		//Check for error after read request
		IF NOT fbADSREADWRITE_ReadAds.BUSY AND NOT fbADSREADWRITE_ReadAds.ERR AND byCounterWaitInStep_ReadAds >= byStaticValueWaitInStep THEN 
			IF udiNumberSizeValues_ReadAds >= 1 AND udiNumberSizeValues_ReadAds <= 4000 THEN
				FOR udiLPCheckErrorAfterReadReq_ReadAds := 1 TO (udiNumberSizeValues_ReadAds * 4) BY 1 DO
					IF arrValueRead_ReadAds[udiLPCheckErrorAfterReadReq_ReadAds] <> 0 THEN iState_ReadAds := 200; EXIT; END_IF
				END_FOR
			END_IF
		END_IF 	
	
		IF NOT fbADSREADWRITE_ReadAds.BUSY AND NOT fbADSREADWRITE_ReadAds.ERR AND byCounterWaitInStep_ReadAds >= byStaticValueWaitInStep AND iState_ReadAds = -5 THEN 
			byCounterWaitInStep_ReadAds := 0;	
				fbADSREADWRITE_ReadAds.WRTRD := FALSE;
				 iState_ReadAds := -4;
				 	udiStartValueReadOutReqBuffer_AdsRead := (udiNumberSizeValues_ReadAds * 4) + 1;	
						udiNumberInProgress_ReadAds := 1;
		 END_IF 
		
			IF FPErrorReadWrite_ReadAds.Q OR timTimout_ReadAds.Q THEN iState_ReadAds := 200; END_IF 	
			
	-4://Copy Value in buffer after read request and clear data
		uiNumberValueSymbolSize_ReadAds := 0; byNumberOfValues_ReadAds_ReadAds := 0; byLenghSymbolName_ReadAds := 0; byValueInTurn_ReadAds := 0; byCounterValue_ReadAds	:= 0;
			uiValueForLoopStart_ReadAds := 0; uiValueForLoopStop_ReadAds := 0; byCounterValueReadOut_ReadAds := 0;
				fbADSREADWRITE_ReadAds.WRTRD := FALSE;	
		arrCounterWriteValueInArray_ReadAds[1] := 0; arrCounterWriteValueInArray_ReadAds[2] := 0; arrCounterWriteValueInArray_ReadAds[3] := 0; arrCounterWriteValueInArray_ReadAds[4] := 0; arrCounterWriteValueInArray_ReadAds[5] := 0;
			arrCounterWriteValueInArray_ReadAds[6] := 0; arrCounterWriteValueInArray_ReadAds[7] := 0; arrCounterWriteValueInArray_ReadAds[8] := 0;
									
		uiCounterArrayOfString_ReadAds := 0;
	
		sStringFloat_ReadAds := ''; iFindPointFloat_ReadAds := 0; iPrecision_ReadAds := 0;
		
		//Copy first 800 default bytes to save resources on small plc's
		MEMCPY(ADR(arrValueAfterRead_ReadAds),ADR(arrValueAfterReadDefault_ReadAds),SIZEOF(arrValueAfterRead_ReadAds));
		
		//Clear lengh from each value
		arrLenghEachValue_ReadAds := arrLenghEachValueDefault_ReadAds;
			
		//Clear array with symbol name and array with the value names
		arrSymbolName_ReadAds := arrSymbolNameDefault_ReadAds;
			arrValueName_ReadAds := arrValueNameDefault_ReadAds; 
	
		//Copy the values
		udiNumberInProgress_ReadAds := LIMIT(1,udiNumberInProgress_ReadAds,10);
			udiStopValueReadOutReqBuffer_AdsRead := (udiStartValueReadOutReqBuffer_AdsRead - 1) + arrInfoValue_Read_Ads[udiNumberInProgress_ReadAds].udiLength;

		IF udiStartValueReadOutReqBuffer_AdsRead >= 1 AND udiStartValueReadOutReqBuffer_AdsRead <= 1600 AND udiStopValueReadOutReqBuffer_AdsRead >= 1 AND udiStopValueReadOutReqBuffer_AdsRead <= 1600 THEN  
			FOR udiLPCopyValueFromReqBuffer_ReadAds := udiStartValueReadOutReqBuffer_AdsRead TO udiStopValueReadOutReqBuffer_AdsRead BY 1 DO
				uiCounterCopyValueFromReqBuffer_ReadAds := LIMIT(1,uiCounterCopyValueFromReqBuffer_ReadAds,1600);	
					arrValueAfterRead_ReadAds[uiCounterCopyValueFromReqBuffer_ReadAds] := arrValueRead_ReadAds[udiLPCopyValueFromReqBuffer_ReadAds]; 
						uiCounterCopyValueFromReqBuffer_ReadAds := uiCounterCopyValueFromReqBuffer_ReadAds + 1;
			END_FOR 
		END_IF		
			
		uiCounterCopyValueFromReqBuffer_ReadAds := 0;
			udiActiveNumberOfSymbol_ReadAds := udiActiveNumberOfSymbol_ReadAds + 1;
				udiActiveNumberOfSymbol_ReadAds := LIMIT(1,udiActiveNumberOfSymbol_ReadAds,Lynus_Standards.Constants_Communicator.udiArraySizeMarkedSymobls);
					udiStartValueReadOutReqBuffer_AdsRead := udiStopValueReadOutReqBuffer_AdsRead + 1;
						iState_ReadAds := -3;
						
	-3://Check whether the write application does not have the same value as when reading
		IF (Lynus_Standards.GVL_Communicator.arrInterfaceInfoAlVariables[byReadWriteArrayNumber,udiActiveNumberOfSymbol_ReadAds].sFullSymbolName <> Lynus_Standards.GVL_Communicator.arrInterfaceInfoValueWriteTo[byReadWriteArrayNumber].sFullSymbolName) 
			// AND m_EnableChange_upload) // Stefan added AND 
			// OR m_TriggerIntervalSend=TRUE THEN 	// STEFAN
			THEN
			iState_ReadAds := 5;
		ELSE
			IF udiActiveNumberOfSymbol_ReadAds < Lynus_Standards.GVL_Communicator.arrCounterVariableInArray[byReadWriteArrayNumber] AND udiNumberInProgress_ReadAds < udiNumberSizeValues_ReadAds THEN iState_ReadAds := -4; udiNumberInProgress_ReadAds := udiNumberInProgress_ReadAds + 1; END_IF
			IF (udiNumberInProgress_ReadAds >= udiNumberSizeValues_ReadAds AND iState_ReadAds = -3) THEN iState_ReadAds := -8; udiNumberInProgress_ReadAds := 0; END_IF
			IF udiActiveNumberOfSymbol_ReadAds >= Lynus_Standards.GVL_Communicator.arrCounterVariableInArray[byReadWriteArrayNumber] THEN iState_ReadAds := -8; udiActiveNumberOfSymbol_ReadAds := 0; udiNumberInProgress_ReadAds := 0; udiRestValueSymbolRead_ReadAds := 0; END_IF 
		END_IF  
	
		//Timeout
		IF timTimout_ReadAds.Q THEN iState_ReadAds := 200; END_IF
		
	5://Write value and symbol name in read array
	
		IF (Lynus_Standards.GVL_Communicator.arrInterfaceInfoAlVariables[byReadWriteArrayNumber,udiActiveNumberOfSymbol_ReadAds].sFullSymbolName <> Lynus_Standards.GVL_Communicator.arrInterfaceInfoValueWriteTo[byReadWriteArrayNumber].sFullSymbolName)
			// AND m_EnableChange_upload) // Stefan added AND 
			// OR m_TriggerIntervalSend=TRUE THEN 	// STEFAN
			THEN
			//Type BOOL
			IF Lynus_Standards.GVL_Communicator.arrInterfaceInfoAlVariables[byReadWriteArrayNumber,udiActiveNumberOfSymbol_ReadAds].sSymbolType = 'BOOL' THEN 
				stADSRead_ReadAds[udiActiveNumberOfSymbol_ReadAds].arrValue := arrValueDefault_ReadAds;
					stADSRead_ReadAds[udiActiveNumberOfSymbol_ReadAds].sFullSymbolName := Lynus_Standards.GVL_Communicator.arrInterfaceInfoAlVariables[byReadWriteArrayNumber,udiActiveNumberOfSymbol_ReadAds].sFullSymbolName; 
						stADSRead_ReadAds[udiActiveNumberOfSymbol_ReadAds].arrValue[1] := BYTE_TO_STRING(arrValueAfterRead_ReadAds[1]); 
			END_IF
				//Type BYTE
				IF Lynus_Standards.GVL_Communicator.arrInterfaceInfoAlVariables[byReadWriteArrayNumber,udiActiveNumberOfSymbol_ReadAds].sSymbolType = 'BYTE' THEN 
					stADSRead_ReadAds[udiActiveNumberOfSymbol_ReadAds].arrValue := arrValueDefault_ReadAds;
						stADSRead_ReadAds[udiActiveNumberOfSymbol_ReadAds].sFullSymbolName := Lynus_Standards.GVL_Communicator.arrInterfaceInfoAlVariables[byReadWriteArrayNumber,udiActiveNumberOfSymbol_ReadAds].sFullSymbolName; 
							stADSRead_ReadAds[udiActiveNumberOfSymbol_ReadAds].arrValue[1] := BYTE_TO_STRING(arrValueAfterRead_ReadAds[1]); 
				END_IF
			//Type WORD
			IF Lynus_Standards.GVL_Communicator.arrInterfaceInfoAlVariables[byReadWriteArrayNumber,udiActiveNumberOfSymbol_ReadAds].sSymbolType = 'WORD' THEN 
				stADSRead_ReadAds[udiActiveNumberOfSymbol_ReadAds].arrValue := arrValueDefault_ReadAds;
					stADSRead_ReadAds[udiActiveNumberOfSymbol_ReadAds].sFullSymbolName := Lynus_Standards.GVL_Communicator.arrInterfaceInfoAlVariables[byReadWriteArrayNumber,udiActiveNumberOfSymbol_ReadAds].sFullSymbolName; 
						stADSRead_ReadAds[udiActiveNumberOfSymbol_ReadAds].arrValue[1] := WORD_TO_STRING(SHL(BYTE_TO_WORD(arrValueAfterRead_ReadAds[2]),8) + BYTE_TO_WORD(arrValueAfterRead_ReadAds[1]));
			END_IF
				//Type DWORD
				IF Lynus_Standards.GVL_Communicator.arrInterfaceInfoAlVariables[byReadWriteArrayNumber,udiActiveNumberOfSymbol_ReadAds].sSymbolType = 'DWORD' THEN 
					stADSRead_ReadAds[udiActiveNumberOfSymbol_ReadAds].arrValue := arrValueDefault_ReadAds;
						stADSRead_ReadAds[udiActiveNumberOfSymbol_ReadAds].sFullSymbolName := Lynus_Standards.GVL_Communicator.arrInterfaceInfoAlVariables[byReadWriteArrayNumber,udiActiveNumberOfSymbol_ReadAds].sFullSymbolName; 
							stADSRead_ReadAds[udiActiveNumberOfSymbol_ReadAds].arrValue[1] := DWORD_TO_STRING(SHL(BYTE_TO_DWORD(arrValueAfterRead_ReadAds[4]),24) + SHL(BYTE_TO_DWORD(arrValueAfterRead_ReadAds[3]),16) + SHL(BYTE_TO_DWORD(arrValueAfterRead_ReadAds[2]),8) + BYTE_TO_DWORD(arrValueAfterRead_ReadAds[1]));
				END_IF
			//Type SINT
			IF Lynus_Standards.GVL_Communicator.arrInterfaceInfoAlVariables[byReadWriteArrayNumber,udiActiveNumberOfSymbol_ReadAds].sSymbolType = 'SINT' THEN 
				stADSRead_ReadAds[udiActiveNumberOfSymbol_ReadAds].arrValue := arrValueDefault_ReadAds;
					stADSRead_ReadAds[udiActiveNumberOfSymbol_ReadAds].sFullSymbolName := Lynus_Standards.GVL_Communicator.arrInterfaceInfoAlVariables[byReadWriteArrayNumber,udiActiveNumberOfSymbol_ReadAds].sFullSymbolName; 
						stADSRead_ReadAds[udiActiveNumberOfSymbol_ReadAds].arrValue[1] := SINT_TO_STRING(BYTE_TO_SINT(arrValueAfterRead_ReadAds[1]));
			END_IF
				//Type USINT
				IF Lynus_Standards.GVL_Communicator.arrInterfaceInfoAlVariables[byReadWriteArrayNumber,udiActiveNumberOfSymbol_ReadAds].sSymbolType = 'USINT' THEN 
					stADSRead_ReadAds[udiActiveNumberOfSymbol_ReadAds].arrValue := arrValueDefault_ReadAds;
						stADSRead_ReadAds[udiActiveNumberOfSymbol_ReadAds].sFullSymbolName := Lynus_Standards.GVL_Communicator.arrInterfaceInfoAlVariables[byReadWriteArrayNumber,udiActiveNumberOfSymbol_ReadAds].sFullSymbolName; 
							stADSRead_ReadAds[udiActiveNumberOfSymbol_ReadAds].arrValue[1] := USINT_TO_STRING(BYTE_TO_USINT(arrValueAfterRead_ReadAds[1]));
				END_IF
			//Type INT
			IF Lynus_Standards.GVL_Communicator.arrInterfaceInfoAlVariables[byReadWriteArrayNumber,udiActiveNumberOfSymbol_ReadAds].sSymbolType = 'INT' THEN 
				stADSRead_ReadAds[udiActiveNumberOfSymbol_ReadAds].arrValue := arrValueDefault_ReadAds;
					stADSRead_ReadAds[udiActiveNumberOfSymbol_ReadAds].sFullSymbolName := Lynus_Standards.GVL_Communicator.arrInterfaceInfoAlVariables[byReadWriteArrayNumber,udiActiveNumberOfSymbol_ReadAds].sFullSymbolName; 
						stADSRead_ReadAds[udiActiveNumberOfSymbol_ReadAds].arrValue[1] := INT_TO_STRING(SHL(BYTE_TO_INT(arrValueAfterRead_ReadAds[2]),8) + BYTE_TO_INT(arrValueAfterRead_ReadAds[1]));
			END_IF
				//Type UINT
				IF Lynus_Standards.GVL_Communicator.arrInterfaceInfoAlVariables[byReadWriteArrayNumber,udiActiveNumberOfSymbol_ReadAds].sSymbolType = 'UINT' THEN 
					stADSRead_ReadAds[udiActiveNumberOfSymbol_ReadAds].arrValue := arrValueDefault_ReadAds;
						stADSRead_ReadAds[udiActiveNumberOfSymbol_ReadAds].sFullSymbolName := Lynus_Standards.GVL_Communicator.arrInterfaceInfoAlVariables[byReadWriteArrayNumber,udiActiveNumberOfSymbol_ReadAds].sFullSymbolName; 
							stADSRead_ReadAds[udiActiveNumberOfSymbol_ReadAds].arrValue[1] := UINT_TO_STRING(SHL(BYTE_TO_UINT(arrValueAfterRead_ReadAds[2]),8) + BYTE_TO_UINT(arrValueAfterRead_ReadAds[1]));
				END_IF
			//Type DINT
			IF Lynus_Standards.GVL_Communicator.arrInterfaceInfoAlVariables[byReadWriteArrayNumber,udiActiveNumberOfSymbol_ReadAds].sSymbolType = 'DINT' THEN 
				stADSRead_ReadAds[udiActiveNumberOfSymbol_ReadAds].arrValue := arrValueDefault_ReadAds;
					stADSRead_ReadAds[udiActiveNumberOfSymbol_ReadAds].sFullSymbolName := Lynus_Standards.GVL_Communicator.arrInterfaceInfoAlVariables[byReadWriteArrayNumber,udiActiveNumberOfSymbol_ReadAds].sFullSymbolName; 
						stADSRead_ReadAds[udiActiveNumberOfSymbol_ReadAds].arrValue[1] := DINT_TO_STRING(SHL(BYTE_TO_DINT(arrValueAfterRead_ReadAds[4]),24) + SHL(BYTE_TO_DINT(arrValueAfterRead_ReadAds[3]),16) + SHL(BYTE_TO_DINT(arrValueAfterRead_ReadAds[2]),8) + BYTE_TO_DINT(arrValueAfterRead_ReadAds[1]));
			END_IF
				//Type UDINT
				IF Lynus_Standards.GVL_Communicator.arrInterfaceInfoAlVariables[byReadWriteArrayNumber,udiActiveNumberOfSymbol_ReadAds].sSymbolType = 'UDINT' THEN 
					stADSRead_ReadAds[udiActiveNumberOfSymbol_ReadAds].arrValue := arrValueDefault_ReadAds;
						stADSRead_ReadAds[udiActiveNumberOfSymbol_ReadAds].sFullSymbolName := Lynus_Standards.GVL_Communicator.arrInterfaceInfoAlVariables[byReadWriteArrayNumber,udiActiveNumberOfSymbol_ReadAds].sFullSymbolName; 
							stADSRead_ReadAds[udiActiveNumberOfSymbol_ReadAds].arrValue[1] := UDINT_TO_STRING(SHL(BYTE_TO_UDINT(arrValueAfterRead_ReadAds[4]),24) + SHL(BYTE_TO_UDINT(arrValueAfterRead_ReadAds[3]),16) + SHL(BYTE_TO_UDINT(arrValueAfterRead_ReadAds[2]),8) + BYTE_TO_UDINT(arrValueAfterRead_ReadAds[1]));
				END_IF
			//Type LINT
			IF Lynus_Standards.GVL_Communicator.arrInterfaceInfoAlVariables[byReadWriteArrayNumber,udiActiveNumberOfSymbol_ReadAds].sSymbolType = 'LINT' THEN 
				stADSRead_ReadAds[udiActiveNumberOfSymbol_ReadAds].arrValue := arrValueDefault_ReadAds;
					stADSRead_ReadAds[udiActiveNumberOfSymbol_ReadAds].sFullSymbolName := Lynus_Standards.GVL_Communicator.arrInterfaceInfoAlVariables[byReadWriteArrayNumber,udiActiveNumberOfSymbol_ReadAds].sFullSymbolName; 
						stADSRead_ReadAds[udiActiveNumberOfSymbol_ReadAds].arrValue[1] := LINT_TO_STRING(SHL(BYTE_TO_LINT(arrValueAfterRead_ReadAds[8]),56) + SHL(BYTE_TO_LINT(arrValueAfterRead_ReadAds[7]),48) + SHL(BYTE_TO_LINT(arrValueAfterRead_ReadAds[6]),40) + SHL(BYTE_TO_LINT(arrValueAfterRead_ReadAds[5]),32) +
																						SHL(BYTE_TO_LINT(arrValueAfterRead_ReadAds[4]),24) + SHL(BYTE_TO_LINT(arrValueAfterRead_ReadAds[3]),16) + SHL(BYTE_TO_LINT(arrValueAfterRead_ReadAds[2]),8) + BYTE_TO_LINT(arrValueAfterRead_ReadAds[1]));
			END_IF
				//Type ULINT
				IF Lynus_Standards.GVL_Communicator.arrInterfaceInfoAlVariables[byReadWriteArrayNumber,udiActiveNumberOfSymbol_ReadAds].sSymbolType = 'ULINT' THEN 
					stADSRead_ReadAds[udiActiveNumberOfSymbol_ReadAds].arrValue := arrValueDefault_ReadAds;
						stADSRead_ReadAds[udiActiveNumberOfSymbol_ReadAds].sFullSymbolName := Lynus_Standards.GVL_Communicator.arrInterfaceInfoAlVariables[byReadWriteArrayNumber,udiActiveNumberOfSymbol_ReadAds].sFullSymbolName; 
							stADSRead_ReadAds[udiActiveNumberOfSymbol_ReadAds].arrValue[1] := ULINT_TO_STRING(SHL(BYTE_TO_ULINT(arrValueAfterRead_ReadAds[8]),56) + SHL(BYTE_TO_ULINT(arrValueAfterRead_ReadAds[7]),48) + SHL(BYTE_TO_ULINT(arrValueAfterRead_ReadAds[6]),40) + SHL(BYTE_TO_ULINT(arrValueAfterRead_ReadAds[5]),32) +
																							SHL(BYTE_TO_ULINT(arrValueAfterRead_ReadAds[4]),24) + SHL(BYTE_TO_ULINT(arrValueAfterRead_ReadAds[3]),16) + SHL(BYTE_TO_ULINT(arrValueAfterRead_ReadAds[2]),8) + BYTE_TO_ULINT(arrValueAfterRead_ReadAds[1]));
				END_IF
			//Type LWORD
			IF Lynus_Standards.GVL_Communicator.arrInterfaceInfoAlVariables[byReadWriteArrayNumber,udiActiveNumberOfSymbol_ReadAds].sSymbolType = 'LWORD' THEN 
				stADSRead_ReadAds[udiActiveNumberOfSymbol_ReadAds].arrValue := arrValueDefault_ReadAds;
					stADSRead_ReadAds[udiActiveNumberOfSymbol_ReadAds].sFullSymbolName := Lynus_Standards.GVL_Communicator.arrInterfaceInfoAlVariables[byReadWriteArrayNumber,udiActiveNumberOfSymbol_ReadAds].sFullSymbolName; 
						stADSRead_ReadAds[udiActiveNumberOfSymbol_ReadAds].arrValue[1] := LWORD_TO_STRING(SHL(BYTE_TO_LWORD(arrValueAfterRead_ReadAds[8]),56) + SHL(BYTE_TO_LWORD(arrValueAfterRead_ReadAds[7]),48) + SHL(BYTE_TO_LWORD(arrValueAfterRead_ReadAds[6]),40) + SHL(BYTE_TO_LWORD(arrValueAfterRead_ReadAds[5]),32) +
																						SHL(BYTE_TO_LWORD(arrValueAfterRead_ReadAds[4]),24) + SHL(BYTE_TO_LWORD(arrValueAfterRead_ReadAds[3]),16) + SHL(BYTE_TO_LWORD(arrValueAfterRead_ReadAds[2]),8) + BYTE_TO_LWORD(arrValueAfterRead_ReadAds[1]));
			END_IF
				//Type REAL
				IF Lynus_Standards.GVL_Communicator.arrInterfaceInfoAlVariables[byReadWriteArrayNumber,udiActiveNumberOfSymbol_ReadAds].sSymbolType = 'REAL' THEN
					stADSRead_ReadAds[udiActiveNumberOfSymbol_ReadAds].arrValue := arrValueDefault_ReadAds;
						stADSRead_ReadAds[udiActiveNumberOfSymbol_ReadAds].sFullSymbolName := Lynus_Standards.GVL_Communicator.arrInterfaceInfoAlVariables[byReadWriteArrayNumber,udiActiveNumberOfSymbol_ReadAds].sFullSymbolName; 	
							unConvertDWORD_TO_REAL_ReadAds.dwRawValue := DINT_TO_DWORD(DWORD_TO_DINT(SHL(BYTE_TO_DWORD(arrValueAfterRead_ReadAds[4]),24) + SHL(BYTE_TO_DWORD(arrValueAfterRead_ReadAds[3]),16) + SHL(BYTE_TO_DWORD(arrValueAfterRead_ReadAds[2]),8) + BYTE_TO_DWORD(arrValueAfterRead_ReadAds[1])));
								IF IsFinite(F_REAL(unConvertDWORD_TO_REAL_ReadAds.rValueFloat)) THEN 
									IF LEN(REAL_TO_STRING(unConvertDWORD_TO_REAL_ReadAds.rValueFloat)) <= 30 THEN 
										IF FIND(REAL_TO_STRING(unConvertDWORD_TO_REAL_ReadAds.rValueFloat),'e') = 0 AND FIND(REAL_TO_STRING(unConvertDWORD_TO_REAL_ReadAds.rValueFloat),'E') = 0 THEN 
											sStringFloat_ReadAds := REAL_TO_STRING(unConvertDWORD_TO_REAL_ReadAds.rValueFloat);
												iFindPointFloat_ReadAds := FIND(sStringFloat_ReadAds,'.');
													sStringFloat_ReadAds := DELETE(sStringFloat_ReadAds,iFindPointFloat_ReadAds,1);
														iPrecision_ReadAds := LEN(sStringFloat_ReadAds);
															iPrecision_ReadAds := LIMIT(0,iPrecision_ReadAds,8);			
											IF LEN(LREAL_TO_FMTSTR(REAL_TO_LREAL(unConvertDWORD_TO_REAL_ReadAds.rValueFloat),iPrecision_ReadAds,TRUE)) <= 30 THEN
												//Check if the output from Function LREAL_TO_FMTSTR is ok 
												IF LREAL_TO_FMTSTR(REAL_TO_LREAL(unConvertDWORD_TO_REAL_ReadAds.rValueFloat),iPrecision_ReadAds,TRUE) <> '#INF' AND LREAL_TO_FMTSTR(REAL_TO_LREAL(unConvertDWORD_TO_REAL_ReadAds.rValueFloat),iPrecision_ReadAds,TRUE) <> '-#INF' AND
													LREAL_TO_FMTSTR(REAL_TO_LREAL(unConvertDWORD_TO_REAL_ReadAds.rValueFloat),iPrecision_ReadAds,TRUE) <> '#QNAN' AND LREAL_TO_FMTSTR(REAL_TO_LREAL(unConvertDWORD_TO_REAL_ReadAds.rValueFloat),iPrecision_ReadAds,TRUE) <> '-#QNAN' AND
														LREAL_TO_FMTSTR(REAL_TO_LREAL(unConvertDWORD_TO_REAL_ReadAds.rValueFloat),iPrecision_ReadAds,TRUE) <> '#OVF' AND LREAL_TO_FMTSTR(REAL_TO_LREAL(unConvertDWORD_TO_REAL_ReadAds.rValueFloat),iPrecision_ReadAds,TRUE) <> '-#OVF' THEN	   	 			
															stADSRead_ReadAds[udiActiveNumberOfSymbol_ReadAds].arrValue[1] := LREAL_TO_FMTSTR(REAL_TO_LREAL(unConvertDWORD_TO_REAL_ReadAds.rValueFloat),iPrecision_ReadAds,TRUE);
												ELSE
													iState_ReadAds := 200;
														uiInternError_ReadAds := 1;
												END_IF
											ELSE
												//Check if the output from Function LREAL_TO_FMTSTR is ok 
												IF MID(LREAL_TO_FMTSTR(REAL_TO_LREAL(unConvertDWORD_TO_REAL_ReadAds.rValueFloat),iPrecision_ReadAds,TRUE),30,1) <> '#INF' AND MID(LREAL_TO_FMTSTR(REAL_TO_LREAL(unConvertDWORD_TO_REAL_ReadAds.rValueFloat),iPrecision_ReadAds,TRUE),30,1) <> '-#INF' AND
													MID(LREAL_TO_FMTSTR(REAL_TO_LREAL(unConvertDWORD_TO_REAL_ReadAds.rValueFloat),iPrecision_ReadAds,TRUE),30,1) <> '#QNAN' AND MID(LREAL_TO_FMTSTR(REAL_TO_LREAL(unConvertDWORD_TO_REAL_ReadAds.rValueFloat),iPrecision_ReadAds,TRUE),30,1) <> '-#QNAN' AND
														MID(LREAL_TO_FMTSTR(REAL_TO_LREAL(unConvertDWORD_TO_REAL_ReadAds.rValueFloat),iPrecision_ReadAds,TRUE),30,1) <> '#OVF' AND MID(LREAL_TO_FMTSTR(REAL_TO_LREAL(unConvertDWORD_TO_REAL_ReadAds.rValueFloat),iPrecision_ReadAds,TRUE),30,1) <> '-#OVF' THEN 
															stADSRead_ReadAds[udiActiveNumberOfSymbol_ReadAds].arrValue[1] := MID(LREAL_TO_FMTSTR(REAL_TO_LREAL(unConvertDWORD_TO_REAL_ReadAds.rValueFloat),iPrecision_ReadAds,TRUE),30,1);
												ELSE
													iState_ReadAds := 200;
														uiInternError_ReadAds := 1;
												END_IF
											END_IF
										ELSE
											stADSRead_ReadAds[udiActiveNumberOfSymbol_ReadAds].arrValue[1] := REAL_TO_STRING(unConvertDWORD_TO_REAL_ReadAds.rValueFloat);
										END_IF 
									ELSE
										iState_ReadAds := 200;
											uiInternError_ReadAds := 1;
									END_IF
								ELSE
									iState_ReadAds := 200;
										uiInternError_ReadAds := 1;	
								END_IF
				END_IF
			//Type LREAL
			IF Lynus_Standards.GVL_Communicator.arrInterfaceInfoAlVariables[byReadWriteArrayNumber,udiActiveNumberOfSymbol_ReadAds].sSymbolType = 'LREAL' THEN
				stADSRead_ReadAds[udiActiveNumberOfSymbol_ReadAds].arrValue := arrValueDefault_ReadAds;
					stADSRead_ReadAds[udiActiveNumberOfSymbol_ReadAds].sFullSymbolName := Lynus_Standards.GVL_Communicator.arrInterfaceInfoAlVariables[byReadWriteArrayNumber,udiActiveNumberOfSymbol_ReadAds].sFullSymbolName; 	
						unConvertULINT_TO_LREAL_ReadAds.uliRawValue := LINT_TO_ULINT(ULINT_TO_LINT(SHL(BYTE_TO_ULINT(arrValueAfterRead_ReadAds[8]),56) + SHL(BYTE_TO_ULINT(arrValueAfterRead_ReadAds[7]),48) + SHL(BYTE_TO_ULINT(arrValueAfterRead_ReadAds[6]),40) + SHL(BYTE_TO_ULINT(arrValueAfterRead_ReadAds[5]),32) +
																		SHL(BYTE_TO_ULINT(arrValueAfterRead_ReadAds[4]),24) + SHL(BYTE_TO_ULINT(arrValueAfterRead_ReadAds[3]),16) + SHL(BYTE_TO_ULINT(arrValueAfterRead_ReadAds[2]),8) + BYTE_TO_ULINT(arrValueAfterRead_ReadAds[1])));
							IF IsFinite(F_LREAL(unConvertULINT_TO_LREAL_ReadAds.lrValueFloat)) THEN
								IF LEN(LREAL_TO_STRING(unConvertULINT_TO_LREAL_ReadAds.lrValueFloat)) <= 30 THEN 
									IF FIND(LREAL_TO_STRING(unConvertULINT_TO_LREAL_ReadAds.lrValueFloat),'e') = 0 AND FIND(LREAL_TO_STRING(unConvertULINT_TO_LREAL_ReadAds.lrValueFloat),'E') = 0 THEN 
										sStringFloat_ReadAds := LREAL_TO_STRING(unConvertULINT_TO_LREAL_ReadAds.lrValueFloat);
											iFindPointFloat_ReadAds := FIND(sStringFloat_ReadAds,'.');
												sStringFloat_ReadAds := DELETE(sStringFloat_ReadAds,iFindPointFloat_ReadAds,1);
													iPrecision_ReadAds := LEN(sStringFloat_ReadAds);
														iPrecision_ReadAds := LIMIT(0,iPrecision_ReadAds,16);
										IF LEN(LREAL_TO_FMTSTR(unConvertULINT_TO_LREAL_ReadAds.lrValueFloat,iPrecision_ReadAds,TRUE)) <= 30 THEN
											//Check if the output from Function LREAL_TO_FMTSTR is ok 
											IF LREAL_TO_FMTSTR(unConvertULINT_TO_LREAL_ReadAds.lrValueFloat,iPrecision_ReadAds,TRUE) <> '#INF' AND LREAL_TO_FMTSTR(unConvertULINT_TO_LREAL_ReadAds.lrValueFloat,iPrecision_ReadAds,TRUE) <> '-#INF' AND
												LREAL_TO_FMTSTR(unConvertULINT_TO_LREAL_ReadAds.lrValueFloat,iPrecision_ReadAds,TRUE) <> '#QNAN' AND LREAL_TO_FMTSTR(unConvertULINT_TO_LREAL_ReadAds.lrValueFloat,iPrecision_ReadAds,TRUE) <> '-#QNAN' AND
													LREAL_TO_FMTSTR(unConvertULINT_TO_LREAL_ReadAds.lrValueFloat,iPrecision_ReadAds,TRUE) <> '#OVF' AND LREAL_TO_FMTSTR(unConvertULINT_TO_LREAL_ReadAds.lrValueFloat,iPrecision_ReadAds,TRUE) <> '-#OVF' THEN
														stADSRead_ReadAds[udiActiveNumberOfSymbol_ReadAds].arrValue[1] := LREAL_TO_FMTSTR(unConvertULINT_TO_LREAL_ReadAds.lrValueFloat,iPrecision_ReadAds,TRUE); 
											ELSE
												iState_ReadAds := 200;
													uiInternError_ReadAds := 1;
											END_IF
										ELSE
											//Check if the output from Function LREAL_TO_FMTSTR is ok 
											IF MID(LREAL_TO_FMTSTR(unConvertULINT_TO_LREAL_ReadAds.lrValueFloat,iPrecision_ReadAds,TRUE),30,1) <> '#INF' AND MID(LREAL_TO_FMTSTR(unConvertULINT_TO_LREAL_ReadAds.lrValueFloat,iPrecision_ReadAds,TRUE),30,1) <> '-#INF' AND
												MID(LREAL_TO_FMTSTR(unConvertULINT_TO_LREAL_ReadAds.lrValueFloat,iPrecision_ReadAds,TRUE),30,1) <> '#QNAN' AND MID(LREAL_TO_FMTSTR(unConvertULINT_TO_LREAL_ReadAds.lrValueFloat,iPrecision_ReadAds,TRUE),30,1) <> '-#QNAN' AND
													MID(LREAL_TO_FMTSTR(unConvertULINT_TO_LREAL_ReadAds.lrValueFloat,iPrecision_ReadAds,TRUE),30,1) <> '#OVF' AND MID(LREAL_TO_FMTSTR(unConvertULINT_TO_LREAL_ReadAds.lrValueFloat,iPrecision_ReadAds,TRUE),30,1) <> '-#OVF' THEN
														stADSRead_ReadAds[udiActiveNumberOfSymbol_ReadAds].arrValue[1] := MID(LREAL_TO_FMTSTR(unConvertULINT_TO_LREAL_ReadAds.lrValueFloat,iPrecision_ReadAds,TRUE),30,1);
											ELSE
												iState_ReadAds := 200;
													uiInternError_ReadAds := 1;
											END_IF 
										END_IF
									ELSE
										stADSRead_ReadAds[udiActiveNumberOfSymbol_ReadAds].arrValue[1] := LREAL_TO_STRING(unConvertULINT_TO_LREAL_ReadAds.lrValueFloat);
									END_IF
								ELSE
									iState_ReadAds := 200;
										uiInternError_ReadAds := 1;
								END_IF
							ELSE
								iState_ReadAds := 200;
									uiInternError_ReadAds := 1;
							END_IF
			END_IF
				//Type STRING(30)
				IF Lynus_Standards.GVL_Communicator.arrInterfaceInfoAlVariables[byReadWriteArrayNumber,udiActiveNumberOfSymbol_ReadAds].sSymbolType = 'STRING(30)' THEN 
					stADSRead_ReadAds[udiActiveNumberOfSymbol_ReadAds].sFullSymbolName := Lynus_Standards.GVL_Communicator.arrInterfaceInfoAlVariables[byReadWriteArrayNumber,udiActiveNumberOfSymbol_ReadAds].sFullSymbolName;
						stADSRead_ReadAds[udiActiveNumberOfSymbol_ReadAds].arrValue := arrValueDefault_ReadAds;
							FOR byLPCheckCharactersAfterReadOut_ReadAds := 1 TO 30 BY 1 DO
								stADSRead_ReadAds[udiActiveNumberOfSymbol_ReadAds].arrValue[1] := CONCAT(stADSRead_ReadAds[udiActiveNumberOfSymbol_ReadAds].arrValue[1],F_ToCHR(arrValueAfterRead_ReadAds[byLPCheckCharactersAfterReadOut_ReadAds]));
									IF arrValueAfterRead_ReadAds[byLPCheckCharactersAfterReadOut_ReadAds] = 0 AND stADSRead_ReadAds[udiActiveNumberOfSymbol_ReadAds].arrValue[1] <> '' THEN 
										EXIT; 
									ELSIF arrValueAfterRead_ReadAds[byLPCheckCharactersAfterReadOut_ReadAds] = 0 AND stADSRead_ReadAds[udiActiveNumberOfSymbol_ReadAds].arrValue[1] = '' THEN 
										stADSRead_ReadAds[udiActiveNumberOfSymbol_ReadAds].arrValue[1] := '#EMPTY#';
											EXIT;	
									END_IF 
							END_FOR		
				END_IF
			//Type TIME and TIME OF DAY
			IF Lynus_Standards.GVL_Communicator.arrInterfaceInfoAlVariables[byReadWriteArrayNumber,udiActiveNumberOfSymbol_ReadAds].sSymbolType = 'TIME' OR Lynus_Standards.GVL_Communicator.arrInterfaceInfoAlVariables[byReadWriteArrayNumber,udiActiveNumberOfSymbol_ReadAds].sSymbolType = 'TIME_OF_DAY' THEN 
				stADSRead_ReadAds[udiActiveNumberOfSymbol_ReadAds].arrValue := arrValueDefault_ReadAds;
					stADSRead_ReadAds[udiActiveNumberOfSymbol_ReadAds].sFullSymbolName := Lynus_Standards.GVL_Communicator.arrInterfaceInfoAlVariables[byReadWriteArrayNumber,udiActiveNumberOfSymbol_ReadAds].sFullSymbolName;
						stADSRead_ReadAds[udiActiveNumberOfSymbol_ReadAds].arrValue[1] := UDINT_TO_STRING(SHL(BYTE_TO_UDINT(arrValueAfterRead_ReadAds[4]),24) + SHL(BYTE_TO_UDINT(arrValueAfterRead_ReadAds[3]),16) + SHL(BYTE_TO_UDINT(arrValueAfterRead_ReadAds[2]),8) + BYTE_TO_UDINT(arrValueAfterRead_ReadAds[1]));	
			END_IF
				//Type DATE and DATE AND TIME
				IF Lynus_Standards.GVL_Communicator.arrInterfaceInfoAlVariables[byReadWriteArrayNumber,udiActiveNumberOfSymbol_ReadAds].sSymbolType = 'DATE' OR Lynus_Standards.GVL_Communicator.arrInterfaceInfoAlVariables[byReadWriteArrayNumber,udiActiveNumberOfSymbol_ReadAds].sSymbolType = 'DATE_AND_TIME' THEN 
					stADSRead_ReadAds[udiActiveNumberOfSymbol_ReadAds].arrValue := arrValueDefault_ReadAds;
						stADSRead_ReadAds[udiActiveNumberOfSymbol_ReadAds].sFullSymbolName := Lynus_Standards.GVL_Communicator.arrInterfaceInfoAlVariables[byReadWriteArrayNumber,udiActiveNumberOfSymbol_ReadAds].sFullSymbolName;
							uliValueDateTime_ReadAds := SHL(BYTE_TO_ULINT(arrValueAfterRead_ReadAds[4]),24) + SHL(BYTE_TO_ULINT(arrValueAfterRead_ReadAds[3]),16) + SHL(BYTE_TO_ULINT(arrValueAfterRead_ReadAds[2]),8) + BYTE_TO_ULINT(arrValueAfterRead_ReadAds[1]);
								uliValueDateTime_ReadAds := uliValueDateTime_ReadAds * 1000;
									stADSRead_ReadAds[udiActiveNumberOfSymbol_ReadAds].arrValue[1] := ULINT_TO_STRING(uliValueDateTime_ReadAds);		
				END_IF
				
			//Type Arrays
			//ARRAY OF BOOL
			IF FIND(Lynus_Standards.GVL_Communicator.arrInterfaceInfoAlVariables[byReadWriteArrayNumber,udiActiveNumberOfSymbol_ReadAds].sSymbolType,'OF BOOL') <> 0 THEN
				stADSRead_ReadAds[udiActiveNumberOfSymbol_ReadAds].sFullSymbolName := Lynus_Standards.GVL_Communicator.arrInterfaceInfoAlVariables[byReadWriteArrayNumber,udiActiveNumberOfSymbol_ReadAds].sFullSymbolName;
					stADSRead_ReadAds[udiActiveNumberOfSymbol_ReadAds].arrValue := arrValueDefault_ReadAds;	
						IF Lynus_Standards.GVL_Communicator.arrInterfaceInfoAlVariables[byReadWriteArrayNumber,udiActiveNumberOfSymbol_ReadAds].uiSizeArray <= Lynus_Standards.Constants_Communicator.bySizeOfValueArray THEN  
							FOR uiLPWriteValueByArray_ReadAds := 1 TO Lynus_Standards.GVL_Communicator.arrInterfaceInfoAlVariables[byReadWriteArrayNumber,udiActiveNumberOfSymbol_ReadAds].uiSizeArray BY 1 DO 	
								stADSRead_ReadAds[udiActiveNumberOfSymbol_ReadAds].arrValue[uiLPWriteValueByArray_ReadAds] := BYTE_TO_STRING(arrValueAfterRead_ReadAds[uiLPWriteValueByArray_ReadAds]);
							END_FOR 
						END_IF
			END_IF 
				//ARRAY OF BYTE
				IF FIND(Lynus_Standards.GVL_Communicator.arrInterfaceInfoAlVariables[byReadWriteArrayNumber,udiActiveNumberOfSymbol_ReadAds].sSymbolType,'OF BYTE') <> 0 THEN
					stADSRead_ReadAds[udiActiveNumberOfSymbol_ReadAds].sFullSymbolName := Lynus_Standards.GVL_Communicator.arrInterfaceInfoAlVariables[byReadWriteArrayNumber,udiActiveNumberOfSymbol_ReadAds].sFullSymbolName;
						stADSRead_ReadAds[udiActiveNumberOfSymbol_ReadAds].arrValue := arrValueDefault_ReadAds;	
							IF Lynus_Standards.GVL_Communicator.arrInterfaceInfoAlVariables[byReadWriteArrayNumber,udiActiveNumberOfSymbol_ReadAds].uiSizeArray <= Lynus_Standards.Constants_Communicator.bySizeOfValueArray THEN  
								FOR uiLPWriteValueByArray_ReadAds := 1 TO Lynus_Standards.GVL_Communicator.arrInterfaceInfoAlVariables[byReadWriteArrayNumber,udiActiveNumberOfSymbol_ReadAds].uiSizeArray BY 1 DO 	
									stADSRead_ReadAds[udiActiveNumberOfSymbol_ReadAds].arrValue[uiLPWriteValueByArray_ReadAds] := BYTE_TO_STRING(arrValueAfterRead_ReadAds[uiLPWriteValueByArray_ReadAds]);
								END_FOR 
							END_IF
				END_IF
			//ARRAY OF WORD
			IF FIND(Lynus_Standards.GVL_Communicator.arrInterfaceInfoAlVariables[byReadWriteArrayNumber,udiActiveNumberOfSymbol_ReadAds].sSymbolType,'OF WORD') <> 0 THEN
				stADSRead_ReadAds[udiActiveNumberOfSymbol_ReadAds].sFullSymbolName := Lynus_Standards.GVL_Communicator.arrInterfaceInfoAlVariables[byReadWriteArrayNumber,udiActiveNumberOfSymbol_ReadAds].sFullSymbolName;
					stADSRead_ReadAds[udiActiveNumberOfSymbol_ReadAds].arrValue := arrValueDefault_ReadAds;	
						IF Lynus_Standards.GVL_Communicator.arrInterfaceInfoAlVariables[byReadWriteArrayNumber,udiActiveNumberOfSymbol_ReadAds].uiSizeArray <= Lynus_Standards.Constants_Communicator.bySizeOfValueArray THEN  
							FOR uiLPWriteValueByArray_ReadAds := 1 TO Lynus_Standards.GVL_Communicator.arrInterfaceInfoAlVariables[byReadWriteArrayNumber,udiActiveNumberOfSymbol_ReadAds].uiSizeArray BY 1 DO
								arrCounterWriteValueInArray_ReadAds[1] := LIMIT(1,arrCounterWriteValueInArray_ReadAds[1],1600); arrCounterWriteValueInArray_ReadAds[2] := LIMIT(2,arrCounterWriteValueInArray_ReadAds[2],1600);
									stADSRead_ReadAds[udiActiveNumberOfSymbol_ReadAds].arrValue[uiLPWriteValueByArray_ReadAds] := WORD_TO_STRING(SHL(BYTE_TO_WORD(arrValueAfterRead_ReadAds[arrCounterWriteValueInArray_ReadAds[2]]),8) + BYTE_TO_WORD(arrValueAfterRead_ReadAds[arrCounterWriteValueInArray_ReadAds[1]]));;
								arrCounterWriteValueInArray_ReadAds[1] := arrCounterWriteValueInArray_ReadAds[1] + 2; arrCounterWriteValueInArray_ReadAds[2] := arrCounterWriteValueInArray_ReadAds[2] + 2;
							END_FOR 
						END_IF
			END_IF
				//ARRAY OF DWORD	
				IF FIND(Lynus_Standards.GVL_Communicator.arrInterfaceInfoAlVariables[byReadWriteArrayNumber,udiActiveNumberOfSymbol_ReadAds].sSymbolType,'OF DWORD') <> 0 THEN
					stADSRead_ReadAds[udiActiveNumberOfSymbol_ReadAds].sFullSymbolName := Lynus_Standards.GVL_Communicator.arrInterfaceInfoAlVariables[byReadWriteArrayNumber,udiActiveNumberOfSymbol_ReadAds].sFullSymbolName;
						stADSRead_ReadAds[udiActiveNumberOfSymbol_ReadAds].arrValue := arrValueDefault_ReadAds;	
							IF Lynus_Standards.GVL_Communicator.arrInterfaceInfoAlVariables[byReadWriteArrayNumber,udiActiveNumberOfSymbol_ReadAds].uiSizeArray <= Lynus_Standards.Constants_Communicator.bySizeOfValueArray THEN  
								FOR uiLPWriteValueByArray_ReadAds := 1 TO Lynus_Standards.GVL_Communicator.arrInterfaceInfoAlVariables[byReadWriteArrayNumber,udiActiveNumberOfSymbol_ReadAds].uiSizeArray BY 1 DO
									arrCounterWriteValueInArray_ReadAds[1] := LIMIT(1,arrCounterWriteValueInArray_ReadAds[1],1600); arrCounterWriteValueInArray_ReadAds[2] := LIMIT(2,arrCounterWriteValueInArray_ReadAds[2],1600);
										arrCounterWriteValueInArray_ReadAds[3] := LIMIT(3,arrCounterWriteValueInArray_ReadAds[3],1600); arrCounterWriteValueInArray_ReadAds[4] := LIMIT(4,arrCounterWriteValueInArray_ReadAds[4],1600);
											stADSRead_ReadAds[udiActiveNumberOfSymbol_ReadAds].arrValue[uiLPWriteValueByArray_ReadAds] := DWORD_TO_STRING(SHL(BYTE_TO_DWORD(arrValueAfterRead_ReadAds[arrCounterWriteValueInArray_ReadAds[4]]),24) + SHL(BYTE_TO_DWORD(arrValueAfterRead_ReadAds[arrCounterWriteValueInArray_ReadAds[3]]),16) + SHL(BYTE_TO_DWORD(arrValueAfterRead_ReadAds[arrCounterWriteValueInArray_ReadAds[2]]),8) + BYTE_TO_DWORD(arrValueAfterRead_ReadAds[arrCounterWriteValueInArray_ReadAds[1]]));
									arrCounterWriteValueInArray_ReadAds[1] := arrCounterWriteValueInArray_ReadAds[1] + 4; arrCounterWriteValueInArray_ReadAds[2] := arrCounterWriteValueInArray_ReadAds[2] + 4;
										arrCounterWriteValueInArray_ReadAds[3] := arrCounterWriteValueInArray_ReadAds[3] + 4; arrCounterWriteValueInArray_ReadAds[4] := arrCounterWriteValueInArray_ReadAds[4] + 4;
								END_FOR 
							END_IF
				END_IF
			//ARRAY OF SINT
			IF FIND(Lynus_Standards.GVL_Communicator.arrInterfaceInfoAlVariables[byReadWriteArrayNumber,udiActiveNumberOfSymbol_ReadAds].sSymbolType,'OF SINT') <> 0 THEN
				stADSRead_ReadAds[udiActiveNumberOfSymbol_ReadAds].sFullSymbolName := Lynus_Standards.GVL_Communicator.arrInterfaceInfoAlVariables[byReadWriteArrayNumber,udiActiveNumberOfSymbol_ReadAds].sFullSymbolName;
					stADSRead_ReadAds[udiActiveNumberOfSymbol_ReadAds].arrValue := arrValueDefault_ReadAds;	
						IF Lynus_Standards.GVL_Communicator.arrInterfaceInfoAlVariables[byReadWriteArrayNumber,udiActiveNumberOfSymbol_ReadAds].uiSizeArray <= Lynus_Standards.Constants_Communicator.bySizeOfValueArray THEN  
							FOR uiLPWriteValueByArray_ReadAds := 1 TO Lynus_Standards.GVL_Communicator.arrInterfaceInfoAlVariables[byReadWriteArrayNumber,udiActiveNumberOfSymbol_ReadAds].uiSizeArray BY 1 DO 	
								stADSRead_ReadAds[udiActiveNumberOfSymbol_ReadAds].arrValue[uiLPWriteValueByArray_ReadAds] := SINT_TO_STRING(BYTE_TO_SINT(arrValueAfterRead_ReadAds[uiLPWriteValueByArray_ReadAds]));
							END_FOR 
						END_IF
			END_IF
				//ARRAY OF USINT
				IF FIND(Lynus_Standards.GVL_Communicator.arrInterfaceInfoAlVariables[byReadWriteArrayNumber,udiActiveNumberOfSymbol_ReadAds].sSymbolType,'OF USINT') <> 0 THEN
					stADSRead_ReadAds[udiActiveNumberOfSymbol_ReadAds].sFullSymbolName := Lynus_Standards.GVL_Communicator.arrInterfaceInfoAlVariables[byReadWriteArrayNumber,udiActiveNumberOfSymbol_ReadAds].sFullSymbolName;
						stADSRead_ReadAds[udiActiveNumberOfSymbol_ReadAds].arrValue := arrValueDefault_ReadAds;	
							IF Lynus_Standards.GVL_Communicator.arrInterfaceInfoAlVariables[byReadWriteArrayNumber,udiActiveNumberOfSymbol_ReadAds].uiSizeArray <= Lynus_Standards.Constants_Communicator.bySizeOfValueArray THEN  
								FOR uiLPWriteValueByArray_ReadAds := 1 TO Lynus_Standards.GVL_Communicator.arrInterfaceInfoAlVariables[byReadWriteArrayNumber,udiActiveNumberOfSymbol_ReadAds].uiSizeArray BY 1 DO 	
									stADSRead_ReadAds[udiActiveNumberOfSymbol_ReadAds].arrValue[uiLPWriteValueByArray_ReadAds] := USINT_TO_STRING(BYTE_TO_USINT(arrValueAfterRead_ReadAds[uiLPWriteValueByArray_ReadAds]));
								END_FOR 
							END_IF
				END_IF
			//ARRAY OF INT
			IF FIND(Lynus_Standards.GVL_Communicator.arrInterfaceInfoAlVariables[byReadWriteArrayNumber,udiActiveNumberOfSymbol_ReadAds].sSymbolType,'OF INT') <> 0 THEN
				stADSRead_ReadAds[udiActiveNumberOfSymbol_ReadAds].sFullSymbolName := Lynus_Standards.GVL_Communicator.arrInterfaceInfoAlVariables[byReadWriteArrayNumber,udiActiveNumberOfSymbol_ReadAds].sFullSymbolName;
					stADSRead_ReadAds[udiActiveNumberOfSymbol_ReadAds].arrValue := arrValueDefault_ReadAds;	
						IF Lynus_Standards.GVL_Communicator.arrInterfaceInfoAlVariables[byReadWriteArrayNumber,udiActiveNumberOfSymbol_ReadAds].uiSizeArray <= Lynus_Standards.Constants_Communicator.bySizeOfValueArray THEN  
							FOR uiLPWriteValueByArray_ReadAds := 1 TO Lynus_Standards.GVL_Communicator.arrInterfaceInfoAlVariables[byReadWriteArrayNumber,udiActiveNumberOfSymbol_ReadAds].uiSizeArray BY 1 DO
								arrCounterWriteValueInArray_ReadAds[1] := LIMIT(1,arrCounterWriteValueInArray_ReadAds[1],1600); arrCounterWriteValueInArray_ReadAds[2] := LIMIT(2,arrCounterWriteValueInArray_ReadAds[2],1600);
									stADSRead_ReadAds[udiActiveNumberOfSymbol_ReadAds].arrValue[uiLPWriteValueByArray_ReadAds] := INT_TO_STRING(SHL(BYTE_TO_INT(arrValueAfterRead_ReadAds[arrCounterWriteValueInArray_ReadAds[2]]),8) + BYTE_TO_INT(arrValueAfterRead_ReadAds[arrCounterWriteValueInArray_ReadAds[1]]));;
								arrCounterWriteValueInArray_ReadAds[1] := arrCounterWriteValueInArray_ReadAds[1] + 2; arrCounterWriteValueInArray_ReadAds[2] := arrCounterWriteValueInArray_ReadAds[2] + 2;
							END_FOR 
						END_IF
			END_IF
				//ARRAY OF UINT
				IF FIND(Lynus_Standards.GVL_Communicator.arrInterfaceInfoAlVariables[byReadWriteArrayNumber,udiActiveNumberOfSymbol_ReadAds].sSymbolType,'OF UINT') <> 0 THEN
					stADSRead_ReadAds[udiActiveNumberOfSymbol_ReadAds].sFullSymbolName := Lynus_Standards.GVL_Communicator.arrInterfaceInfoAlVariables[byReadWriteArrayNumber,udiActiveNumberOfSymbol_ReadAds].sFullSymbolName;
						stADSRead_ReadAds[udiActiveNumberOfSymbol_ReadAds].arrValue := arrValueDefault_ReadAds;	
							IF Lynus_Standards.GVL_Communicator.arrInterfaceInfoAlVariables[byReadWriteArrayNumber,udiActiveNumberOfSymbol_ReadAds].uiSizeArray <= Lynus_Standards.Constants_Communicator.bySizeOfValueArray THEN  
								FOR uiLPWriteValueByArray_ReadAds := 1 TO Lynus_Standards.GVL_Communicator.arrInterfaceInfoAlVariables[byReadWriteArrayNumber,udiActiveNumberOfSymbol_ReadAds].uiSizeArray BY 1 DO
									arrCounterWriteValueInArray_ReadAds[1] := LIMIT(1,arrCounterWriteValueInArray_ReadAds[1],1600); arrCounterWriteValueInArray_ReadAds[2] := LIMIT(2,arrCounterWriteValueInArray_ReadAds[2],1600);
										stADSRead_ReadAds[udiActiveNumberOfSymbol_ReadAds].arrValue[uiLPWriteValueByArray_ReadAds] := UINT_TO_STRING(SHL(BYTE_TO_UINT(arrValueAfterRead_ReadAds[arrCounterWriteValueInArray_ReadAds[2]]),8) + BYTE_TO_UINT(arrValueAfterRead_ReadAds[arrCounterWriteValueInArray_ReadAds[1]]));;
									arrCounterWriteValueInArray_ReadAds[1] := arrCounterWriteValueInArray_ReadAds[1] + 2; arrCounterWriteValueInArray_ReadAds[2] := arrCounterWriteValueInArray_ReadAds[2] + 2;
								END_FOR 
							END_IF
				END_IF
			//ARRAY OF DINT	
			IF FIND(Lynus_Standards.GVL_Communicator.arrInterfaceInfoAlVariables[byReadWriteArrayNumber,udiActiveNumberOfSymbol_ReadAds].sSymbolType,'OF DINT') <> 0 THEN
				stADSRead_ReadAds[udiActiveNumberOfSymbol_ReadAds].sFullSymbolName := Lynus_Standards.GVL_Communicator.arrInterfaceInfoAlVariables[byReadWriteArrayNumber,udiActiveNumberOfSymbol_ReadAds].sFullSymbolName;
					stADSRead_ReadAds[udiActiveNumberOfSymbol_ReadAds].arrValue := arrValueDefault_ReadAds;	
						IF Lynus_Standards.GVL_Communicator.arrInterfaceInfoAlVariables[byReadWriteArrayNumber,udiActiveNumberOfSymbol_ReadAds].uiSizeArray <= Lynus_Standards.Constants_Communicator.bySizeOfValueArray THEN  
							FOR uiLPWriteValueByArray_ReadAds := 1 TO Lynus_Standards.GVL_Communicator.arrInterfaceInfoAlVariables[byReadWriteArrayNumber,udiActiveNumberOfSymbol_ReadAds].uiSizeArray BY 1 DO
								arrCounterWriteValueInArray_ReadAds[1] := LIMIT(1,arrCounterWriteValueInArray_ReadAds[1],1600); arrCounterWriteValueInArray_ReadAds[2] := LIMIT(2,arrCounterWriteValueInArray_ReadAds[2],1600);
									arrCounterWriteValueInArray_ReadAds[3] := LIMIT(3,arrCounterWriteValueInArray_ReadAds[3],1600); arrCounterWriteValueInArray_ReadAds[4] := LIMIT(4,arrCounterWriteValueInArray_ReadAds[4],1600);
										stADSRead_ReadAds[udiActiveNumberOfSymbol_ReadAds].arrValue[uiLPWriteValueByArray_ReadAds] := DINT_TO_STRING(SHL(BYTE_TO_DINT(arrValueAfterRead_ReadAds[arrCounterWriteValueInArray_ReadAds[4]]),24) + SHL(BYTE_TO_DINT(arrValueAfterRead_ReadAds[arrCounterWriteValueInArray_ReadAds[3]]),16) + SHL(BYTE_TO_DINT(arrValueAfterRead_ReadAds[arrCounterWriteValueInArray_ReadAds[2]]),8) + BYTE_TO_DINT(arrValueAfterRead_ReadAds[arrCounterWriteValueInArray_ReadAds[1]]));
								arrCounterWriteValueInArray_ReadAds[1] := arrCounterWriteValueInArray_ReadAds[1] + 4; arrCounterWriteValueInArray_ReadAds[2] := arrCounterWriteValueInArray_ReadAds[2] + 4;
									arrCounterWriteValueInArray_ReadAds[3] := arrCounterWriteValueInArray_ReadAds[3] + 4; arrCounterWriteValueInArray_ReadAds[4] := arrCounterWriteValueInArray_ReadAds[4] + 4;
							END_FOR 
						END_IF
			END_IF
				//ARRAY OF UDINT	
				IF FIND(Lynus_Standards.GVL_Communicator.arrInterfaceInfoAlVariables[byReadWriteArrayNumber,udiActiveNumberOfSymbol_ReadAds].sSymbolType,'OF UDINT') <> 0 THEN
					stADSRead_ReadAds[udiActiveNumberOfSymbol_ReadAds].sFullSymbolName := Lynus_Standards.GVL_Communicator.arrInterfaceInfoAlVariables[byReadWriteArrayNumber,udiActiveNumberOfSymbol_ReadAds].sFullSymbolName;
						stADSRead_ReadAds[udiActiveNumberOfSymbol_ReadAds].arrValue := arrValueDefault_ReadAds;	
							IF Lynus_Standards.GVL_Communicator.arrInterfaceInfoAlVariables[byReadWriteArrayNumber,udiActiveNumberOfSymbol_ReadAds].uiSizeArray <= Lynus_Standards.Constants_Communicator.bySizeOfValueArray THEN  
								FOR uiLPWriteValueByArray_ReadAds := 1 TO Lynus_Standards.GVL_Communicator.arrInterfaceInfoAlVariables[byReadWriteArrayNumber,udiActiveNumberOfSymbol_ReadAds].uiSizeArray BY 1 DO
									arrCounterWriteValueInArray_ReadAds[1] := LIMIT(1,arrCounterWriteValueInArray_ReadAds[1],1600); arrCounterWriteValueInArray_ReadAds[2] := LIMIT(2,arrCounterWriteValueInArray_ReadAds[2],1600);
										arrCounterWriteValueInArray_ReadAds[3] := LIMIT(3,arrCounterWriteValueInArray_ReadAds[3],1600); arrCounterWriteValueInArray_ReadAds[4] := LIMIT(4,arrCounterWriteValueInArray_ReadAds[4],1600);
											stADSRead_ReadAds[udiActiveNumberOfSymbol_ReadAds].arrValue[uiLPWriteValueByArray_ReadAds] := UDINT_TO_STRING(SHL(BYTE_TO_UDINT(arrValueAfterRead_ReadAds[arrCounterWriteValueInArray_ReadAds[4]]),24) + SHL(BYTE_TO_UDINT(arrValueAfterRead_ReadAds[arrCounterWriteValueInArray_ReadAds[3]]),16) + SHL(BYTE_TO_UDINT(arrValueAfterRead_ReadAds[arrCounterWriteValueInArray_ReadAds[2]]),8) + BYTE_TO_UDINT(arrValueAfterRead_ReadAds[arrCounterWriteValueInArray_ReadAds[1]]));
									arrCounterWriteValueInArray_ReadAds[1] := arrCounterWriteValueInArray_ReadAds[1] + 4; arrCounterWriteValueInArray_ReadAds[2] := arrCounterWriteValueInArray_ReadAds[2] + 4;
										arrCounterWriteValueInArray_ReadAds[3] := arrCounterWriteValueInArray_ReadAds[3] + 4; arrCounterWriteValueInArray_ReadAds[4] := arrCounterWriteValueInArray_ReadAds[4] + 4;
								END_FOR 
							END_IF
				END_IF
					//ARRAY OF LINT	
					IF FIND(Lynus_Standards.GVL_Communicator.arrInterfaceInfoAlVariables[byReadWriteArrayNumber,udiActiveNumberOfSymbol_ReadAds].sSymbolType,'OF LINT') <> 0 THEN
						stADSRead_ReadAds[udiActiveNumberOfSymbol_ReadAds].sFullSymbolName := Lynus_Standards.GVL_Communicator.arrInterfaceInfoAlVariables[byReadWriteArrayNumber,udiActiveNumberOfSymbol_ReadAds].sFullSymbolName;
							stADSRead_ReadAds[udiActiveNumberOfSymbol_ReadAds].arrValue := arrValueDefault_ReadAds;	
								IF Lynus_Standards.GVL_Communicator.arrInterfaceInfoAlVariables[byReadWriteArrayNumber,udiActiveNumberOfSymbol_ReadAds].uiSizeArray <= Lynus_Standards.Constants_Communicator.bySizeOfValueArray THEN  
									FOR uiLPWriteValueByArray_ReadAds := 1 TO Lynus_Standards.GVL_Communicator.arrInterfaceInfoAlVariables[byReadWriteArrayNumber,udiActiveNumberOfSymbol_ReadAds].uiSizeArray BY 1 DO
										arrCounterWriteValueInArray_ReadAds[1] := LIMIT(1,arrCounterWriteValueInArray_ReadAds[1],1600); arrCounterWriteValueInArray_ReadAds[2] := LIMIT(2,arrCounterWriteValueInArray_ReadAds[2],1600);
											arrCounterWriteValueInArray_ReadAds[3] := LIMIT(3,arrCounterWriteValueInArray_ReadAds[3],1600); arrCounterWriteValueInArray_ReadAds[4] := LIMIT(4,arrCounterWriteValueInArray_ReadAds[4],1600);
												arrCounterWriteValueInArray_ReadAds[5] := LIMIT(5,arrCounterWriteValueInArray_ReadAds[5],1600); arrCounterWriteValueInArray_ReadAds[6] := LIMIT(6,arrCounterWriteValueInArray_ReadAds[6],1600);
													arrCounterWriteValueInArray_ReadAds[7] := LIMIT(7,arrCounterWriteValueInArray_ReadAds[7],1600); arrCounterWriteValueInArray_ReadAds[8] := LIMIT(8,arrCounterWriteValueInArray_ReadAds[8],1600);
														stADSRead_ReadAds[udiActiveNumberOfSymbol_ReadAds].arrValue[uiLPWriteValueByArray_ReadAds] := LINT_TO_STRING(SHL(BYTE_TO_LINT(arrValueAfterRead_ReadAds[arrCounterWriteValueInArray_ReadAds[8]]),56) + SHL(BYTE_TO_LINT(arrValueAfterRead_ReadAds[arrCounterWriteValueInArray_ReadAds[7]]),48) + SHL(BYTE_TO_LINT(arrValueAfterRead_ReadAds[arrCounterWriteValueInArray_ReadAds[6]]),40) + SHL(BYTE_TO_LINT(arrValueAfterRead_ReadAds[arrCounterWriteValueInArray_ReadAds[5]]),32) +
																																							SHL(BYTE_TO_LINT(arrValueAfterRead_ReadAds[arrCounterWriteValueInArray_ReadAds[4]]),24) + SHL(BYTE_TO_LINT(arrValueAfterRead_ReadAds[arrCounterWriteValueInArray_ReadAds[3]]),16) + SHL(BYTE_TO_LINT(arrValueAfterRead_ReadAds[arrCounterWriteValueInArray_ReadAds[2]]),8) + BYTE_TO_LINT(arrValueAfterRead_ReadAds[arrCounterWriteValueInArray_ReadAds[1]]));
										arrCounterWriteValueInArray_ReadAds[1] := arrCounterWriteValueInArray_ReadAds[1] + 8; arrCounterWriteValueInArray_ReadAds[2] := arrCounterWriteValueInArray_ReadAds[2] + 8;
											arrCounterWriteValueInArray_ReadAds[3] := arrCounterWriteValueInArray_ReadAds[3] + 8; arrCounterWriteValueInArray_ReadAds[4] := arrCounterWriteValueInArray_ReadAds[4] + 8;
												arrCounterWriteValueInArray_ReadAds[5] := arrCounterWriteValueInArray_ReadAds[5] + 8; arrCounterWriteValueInArray_ReadAds[6] := arrCounterWriteValueInArray_ReadAds[6] + 8;
													arrCounterWriteValueInArray_ReadAds[7] := arrCounterWriteValueInArray_ReadAds[7] + 8; arrCounterWriteValueInArray_ReadAds[8] := arrCounterWriteValueInArray_ReadAds[8] + 8;
									END_FOR 
								END_IF
					END_IF
				//ARRAY OF ULINT	
				IF FIND(Lynus_Standards.GVL_Communicator.arrInterfaceInfoAlVariables[byReadWriteArrayNumber,udiActiveNumberOfSymbol_ReadAds].sSymbolType,'OF ULINT') <> 0 THEN
					stADSRead_ReadAds[udiActiveNumberOfSymbol_ReadAds].sFullSymbolName := Lynus_Standards.GVL_Communicator.arrInterfaceInfoAlVariables[byReadWriteArrayNumber,udiActiveNumberOfSymbol_ReadAds].sFullSymbolName;
						stADSRead_ReadAds[udiActiveNumberOfSymbol_ReadAds].arrValue := arrValueDefault_ReadAds;	
							IF Lynus_Standards.GVL_Communicator.arrInterfaceInfoAlVariables[byReadWriteArrayNumber,udiActiveNumberOfSymbol_ReadAds].uiSizeArray <= Lynus_Standards.Constants_Communicator.bySizeOfValueArray THEN  
								FOR uiLPWriteValueByArray_ReadAds := 1 TO Lynus_Standards.GVL_Communicator.arrInterfaceInfoAlVariables[byReadWriteArrayNumber,udiActiveNumberOfSymbol_ReadAds].uiSizeArray BY 1 DO
									arrCounterWriteValueInArray_ReadAds[1] := LIMIT(1,arrCounterWriteValueInArray_ReadAds[1],1600); arrCounterWriteValueInArray_ReadAds[2] := LIMIT(2,arrCounterWriteValueInArray_ReadAds[2],1600);
										arrCounterWriteValueInArray_ReadAds[3] := LIMIT(3,arrCounterWriteValueInArray_ReadAds[3],1600); arrCounterWriteValueInArray_ReadAds[4] := LIMIT(4,arrCounterWriteValueInArray_ReadAds[4],1600);
											arrCounterWriteValueInArray_ReadAds[5] := LIMIT(5,arrCounterWriteValueInArray_ReadAds[5],1600); arrCounterWriteValueInArray_ReadAds[6] := LIMIT(6,arrCounterWriteValueInArray_ReadAds[6],1600);
												arrCounterWriteValueInArray_ReadAds[7] := LIMIT(7,arrCounterWriteValueInArray_ReadAds[7],1600); arrCounterWriteValueInArray_ReadAds[8] := LIMIT(8,arrCounterWriteValueInArray_ReadAds[8],1600);
													stADSRead_ReadAds[udiActiveNumberOfSymbol_ReadAds].arrValue[uiLPWriteValueByArray_ReadAds] := ULINT_TO_STRING(SHL(BYTE_TO_ULINT(arrValueAfterRead_ReadAds[arrCounterWriteValueInArray_ReadAds[8]]),56) + SHL(BYTE_TO_ULINT(arrValueAfterRead_ReadAds[arrCounterWriteValueInArray_ReadAds[7]]),48) + SHL(BYTE_TO_ULINT(arrValueAfterRead_ReadAds[arrCounterWriteValueInArray_ReadAds[6]]),40) + SHL(BYTE_TO_ULINT(arrValueAfterRead_ReadAds[arrCounterWriteValueInArray_ReadAds[5]]),32) +
																																						SHL(BYTE_TO_ULINT(arrValueAfterRead_ReadAds[arrCounterWriteValueInArray_ReadAds[4]]),24) + SHL(BYTE_TO_ULINT(arrValueAfterRead_ReadAds[arrCounterWriteValueInArray_ReadAds[3]]),16) + SHL(BYTE_TO_ULINT(arrValueAfterRead_ReadAds[arrCounterWriteValueInArray_ReadAds[2]]),8) + BYTE_TO_ULINT(arrValueAfterRead_ReadAds[arrCounterWriteValueInArray_ReadAds[1]]));
									arrCounterWriteValueInArray_ReadAds[1] := arrCounterWriteValueInArray_ReadAds[1] + 8; arrCounterWriteValueInArray_ReadAds[2] := arrCounterWriteValueInArray_ReadAds[2] + 8;
										arrCounterWriteValueInArray_ReadAds[3] := arrCounterWriteValueInArray_ReadAds[3] + 8; arrCounterWriteValueInArray_ReadAds[4] := arrCounterWriteValueInArray_ReadAds[4] + 8;
											arrCounterWriteValueInArray_ReadAds[5] := arrCounterWriteValueInArray_ReadAds[5] + 8; arrCounterWriteValueInArray_ReadAds[6] := arrCounterWriteValueInArray_ReadAds[6] + 8;
												arrCounterWriteValueInArray_ReadAds[7] := arrCounterWriteValueInArray_ReadAds[7] + 8; arrCounterWriteValueInArray_ReadAds[8] := arrCounterWriteValueInArray_ReadAds[8] + 8;
								END_FOR 
							END_IF
				END_IF
					//ARRAY OF LWORD	
					IF FIND(Lynus_Standards.GVL_Communicator.arrInterfaceInfoAlVariables[byReadWriteArrayNumber,udiActiveNumberOfSymbol_ReadAds].sSymbolType,'OF LWORD') <> 0 THEN
						stADSRead_ReadAds[udiActiveNumberOfSymbol_ReadAds].sFullSymbolName := Lynus_Standards.GVL_Communicator.arrInterfaceInfoAlVariables[byReadWriteArrayNumber,udiActiveNumberOfSymbol_ReadAds].sFullSymbolName;
							stADSRead_ReadAds[udiActiveNumberOfSymbol_ReadAds].arrValue := arrValueDefault_ReadAds;	
								IF Lynus_Standards.GVL_Communicator.arrInterfaceInfoAlVariables[byReadWriteArrayNumber,udiActiveNumberOfSymbol_ReadAds].uiSizeArray <= Lynus_Standards.Constants_Communicator.bySizeOfValueArray THEN  
									FOR uiLPWriteValueByArray_ReadAds := 1 TO Lynus_Standards.GVL_Communicator.arrInterfaceInfoAlVariables[byReadWriteArrayNumber,udiActiveNumberOfSymbol_ReadAds].uiSizeArray BY 1 DO
										arrCounterWriteValueInArray_ReadAds[1] := LIMIT(1,arrCounterWriteValueInArray_ReadAds[1],1600); arrCounterWriteValueInArray_ReadAds[2] := LIMIT(2,arrCounterWriteValueInArray_ReadAds[2],1600);
											arrCounterWriteValueInArray_ReadAds[3] := LIMIT(3,arrCounterWriteValueInArray_ReadAds[3],1600); arrCounterWriteValueInArray_ReadAds[4] := LIMIT(4,arrCounterWriteValueInArray_ReadAds[4],1600);
												arrCounterWriteValueInArray_ReadAds[5] := LIMIT(5,arrCounterWriteValueInArray_ReadAds[5],1600); arrCounterWriteValueInArray_ReadAds[6] := LIMIT(6,arrCounterWriteValueInArray_ReadAds[6],1600);
													arrCounterWriteValueInArray_ReadAds[7] := LIMIT(7,arrCounterWriteValueInArray_ReadAds[7],1600); arrCounterWriteValueInArray_ReadAds[8] := LIMIT(8,arrCounterWriteValueInArray_ReadAds[8],1600);
														stADSRead_ReadAds[udiActiveNumberOfSymbol_ReadAds].arrValue[uiLPWriteValueByArray_ReadAds] := LWORD_TO_STRING(SHL(BYTE_TO_LWORD(arrValueAfterRead_ReadAds[arrCounterWriteValueInArray_ReadAds[8]]),56) + SHL(BYTE_TO_LWORD(arrValueAfterRead_ReadAds[arrCounterWriteValueInArray_ReadAds[7]]),48) + SHL(BYTE_TO_LWORD(arrValueAfterRead_ReadAds[arrCounterWriteValueInArray_ReadAds[6]]),40) + SHL(BYTE_TO_LWORD(arrValueAfterRead_ReadAds[arrCounterWriteValueInArray_ReadAds[5]]),32) +
																																							SHL(BYTE_TO_LWORD(arrValueAfterRead_ReadAds[arrCounterWriteValueInArray_ReadAds[4]]),24) + SHL(BYTE_TO_LWORD(arrValueAfterRead_ReadAds[arrCounterWriteValueInArray_ReadAds[3]]),16) + SHL(BYTE_TO_LWORD(arrValueAfterRead_ReadAds[arrCounterWriteValueInArray_ReadAds[2]]),8) + BYTE_TO_LWORD(arrValueAfterRead_ReadAds[arrCounterWriteValueInArray_ReadAds[1]]));
										arrCounterWriteValueInArray_ReadAds[1] := arrCounterWriteValueInArray_ReadAds[1] + 8; arrCounterWriteValueInArray_ReadAds[2] := arrCounterWriteValueInArray_ReadAds[2] + 8;
											arrCounterWriteValueInArray_ReadAds[3] := arrCounterWriteValueInArray_ReadAds[3] + 8; arrCounterWriteValueInArray_ReadAds[4] := arrCounterWriteValueInArray_ReadAds[4] + 8;
												arrCounterWriteValueInArray_ReadAds[5] := arrCounterWriteValueInArray_ReadAds[5] + 8; arrCounterWriteValueInArray_ReadAds[6] := arrCounterWriteValueInArray_ReadAds[6] + 8;
													arrCounterWriteValueInArray_ReadAds[7] := arrCounterWriteValueInArray_ReadAds[7] + 8; arrCounterWriteValueInArray_ReadAds[8] := arrCounterWriteValueInArray_ReadAds[8] + 8;
									END_FOR 
								END_IF
					END_IF
				//ARRAY OF REAL
				IF FIND(Lynus_Standards.GVL_Communicator.arrInterfaceInfoAlVariables[byReadWriteArrayNumber,udiActiveNumberOfSymbol_ReadAds].sSymbolType,'OF REAL') <> 0 THEN
					stADSRead_ReadAds[udiActiveNumberOfSymbol_ReadAds].sFullSymbolName := Lynus_Standards.GVL_Communicator.arrInterfaceInfoAlVariables[byReadWriteArrayNumber,udiActiveNumberOfSymbol_ReadAds].sFullSymbolName;
						stADSRead_ReadAds[udiActiveNumberOfSymbol_ReadAds].arrValue := arrValueDefault_ReadAds;	
							IF Lynus_Standards.GVL_Communicator.arrInterfaceInfoAlVariables[byReadWriteArrayNumber,udiActiveNumberOfSymbol_ReadAds].uiSizeArray <= Lynus_Standards.Constants_Communicator.bySizeOfValueArray THEN  
								FOR uiLPWriteValueByArray_ReadAds := 1 TO Lynus_Standards.GVL_Communicator.arrInterfaceInfoAlVariables[byReadWriteArrayNumber,udiActiveNumberOfSymbol_ReadAds].uiSizeArray BY 1 DO
									arrCounterWriteValueInArray_ReadAds[1] := LIMIT(1,arrCounterWriteValueInArray_ReadAds[1],1600); arrCounterWriteValueInArray_ReadAds[2] := LIMIT(2,arrCounterWriteValueInArray_ReadAds[2],1600);
										arrCounterWriteValueInArray_ReadAds[3] := LIMIT(3,arrCounterWriteValueInArray_ReadAds[3],1600); arrCounterWriteValueInArray_ReadAds[4] := LIMIT(4,arrCounterWriteValueInArray_ReadAds[4],1600);
											unConvertDWORD_TO_REAL_ReadAds.dwRawValue := DINT_TO_DWORD(DWORD_TO_DINT(SHL(BYTE_TO_DWORD(arrValueAfterRead_ReadAds[arrCounterWriteValueInArray_ReadAds[4]]),24) + SHL(BYTE_TO_DWORD(arrValueAfterRead_ReadAds[arrCounterWriteValueInArray_ReadAds[3]]),16) + SHL(BYTE_TO_DWORD(arrValueAfterRead_ReadAds[arrCounterWriteValueInArray_ReadAds[2]]),8) + BYTE_TO_DWORD(arrValueAfterRead_ReadAds[arrCounterWriteValueInArray_ReadAds[1]])));
									arrCounterWriteValueInArray_ReadAds[1] := arrCounterWriteValueInArray_ReadAds[1] + 4; arrCounterWriteValueInArray_ReadAds[2] := arrCounterWriteValueInArray_ReadAds[2] + 4;
										arrCounterWriteValueInArray_ReadAds[3] := arrCounterWriteValueInArray_ReadAds[3] + 4; arrCounterWriteValueInArray_ReadAds[4] := arrCounterWriteValueInArray_ReadAds[4] + 4;					
											IF IsFinite(F_REAL(unConvertDWORD_TO_REAL_ReadAds.rValueFloat)) THEN 
												IF LEN(REAL_TO_STRING(unConvertDWORD_TO_REAL_ReadAds.rValueFloat)) <= 30 THEN 
													IF FIND(REAL_TO_STRING(unConvertDWORD_TO_REAL_ReadAds.rValueFloat),'e') = 0 AND FIND(REAL_TO_STRING(unConvertDWORD_TO_REAL_ReadAds.rValueFloat),'E') = 0 THEN 
														sStringFloat_ReadAds := REAL_TO_STRING(unConvertDWORD_TO_REAL_ReadAds.rValueFloat);
															iFindPointFloat_ReadAds := FIND(sStringFloat_ReadAds,'.');
																sStringFloat_ReadAds := DELETE(sStringFloat_ReadAds,iFindPointFloat_ReadAds,1);
																	iPrecision_ReadAds := LEN(sStringFloat_ReadAds);
																		iPrecision_ReadAds := LIMIT(0,iPrecision_ReadAds,8);
														IF LEN(LREAL_TO_FMTSTR(REAL_TO_LREAL(unConvertDWORD_TO_REAL_ReadAds.rValueFloat),iPrecision_ReadAds,TRUE)) <= 30 THEN	 			
															//Check if the output from Function LREAL_TO_FMTSTR is ok 
															IF LREAL_TO_FMTSTR(REAL_TO_LREAL(unConvertDWORD_TO_REAL_ReadAds.rValueFloat),iPrecision_ReadAds,TRUE) <> '#INF' AND LREAL_TO_FMTSTR(REAL_TO_LREAL(unConvertDWORD_TO_REAL_ReadAds.rValueFloat),iPrecision_ReadAds,TRUE) <> '-#INF' AND
																LREAL_TO_FMTSTR(REAL_TO_LREAL(unConvertDWORD_TO_REAL_ReadAds.rValueFloat),iPrecision_ReadAds,TRUE) <> '#QNAN' AND LREAL_TO_FMTSTR(REAL_TO_LREAL(unConvertDWORD_TO_REAL_ReadAds.rValueFloat),iPrecision_ReadAds,TRUE) <> '-#QNAN' AND
																	LREAL_TO_FMTSTR(REAL_TO_LREAL(unConvertDWORD_TO_REAL_ReadAds.rValueFloat),iPrecision_ReadAds,TRUE) <> '#OVF' AND LREAL_TO_FMTSTR(REAL_TO_LREAL(unConvertDWORD_TO_REAL_ReadAds.rValueFloat),iPrecision_ReadAds,TRUE) <> '-#OVF' THEN	   	 			
																		stADSRead_ReadAds[udiActiveNumberOfSymbol_ReadAds].arrValue[uiLPWriteValueByArray_ReadAds] := LREAL_TO_FMTSTR(REAL_TO_LREAL(unConvertDWORD_TO_REAL_ReadAds.rValueFloat),iPrecision_ReadAds,TRUE);
															ELSE
																iState_ReadAds := 200;
																	uiInternError_ReadAds := 1;
															END_IF
														ELSE
															//Check if the output from Function LREAL_TO_FMTSTR is ok 
															IF MID(LREAL_TO_FMTSTR(REAL_TO_LREAL(unConvertDWORD_TO_REAL_ReadAds.rValueFloat),iPrecision_ReadAds,TRUE),30,1) <> '#INF' AND MID(LREAL_TO_FMTSTR(REAL_TO_LREAL(unConvertDWORD_TO_REAL_ReadAds.rValueFloat),iPrecision_ReadAds,TRUE),30,1) <> '-#INF' AND
																MID(LREAL_TO_FMTSTR(REAL_TO_LREAL(unConvertDWORD_TO_REAL_ReadAds.rValueFloat),iPrecision_ReadAds,TRUE),30,1) <> '#QNAN' AND MID(LREAL_TO_FMTSTR(REAL_TO_LREAL(unConvertDWORD_TO_REAL_ReadAds.rValueFloat),iPrecision_ReadAds,TRUE),30,1) <> '-#QNAN' AND
																	MID(LREAL_TO_FMTSTR(REAL_TO_LREAL(unConvertDWORD_TO_REAL_ReadAds.rValueFloat),iPrecision_ReadAds,TRUE),30,1) <> '#OVF' AND MID(LREAL_TO_FMTSTR(REAL_TO_LREAL(unConvertDWORD_TO_REAL_ReadAds.rValueFloat),iPrecision_ReadAds,TRUE),30,1) <> '-#OVF' THEN 
																		stADSRead_ReadAds[udiActiveNumberOfSymbol_ReadAds].arrValue[uiLPWriteValueByArray_ReadAds] := MID(LREAL_TO_FMTSTR(REAL_TO_LREAL(unConvertDWORD_TO_REAL_ReadAds.rValueFloat),iPrecision_ReadAds,TRUE),30,1);
															ELSE
																iState_ReadAds := 200;
																	uiInternError_ReadAds := 1;
															END_IF
														END_IF
													ELSE
														stADSRead_ReadAds[udiActiveNumberOfSymbol_ReadAds].arrValue[uiLPWriteValueByArray_ReadAds] := REAL_TO_STRING(unConvertDWORD_TO_REAL_ReadAds.rValueFloat);
													END_IF 
												ELSE
													iState_ReadAds := 200;
														uiInternError_ReadAds := 1;
												END_IF
											ELSE
												iState_ReadAds := 200;
													uiInternError_ReadAds := 1;	
											END_IF
								END_FOR 
							END_IF
				END_IF
					//ARRAY OF LREAL
					IF FIND(Lynus_Standards.GVL_Communicator.arrInterfaceInfoAlVariables[byReadWriteArrayNumber,udiActiveNumberOfSymbol_ReadAds].sSymbolType,'OF LREAL') <> 0 THEN
						stADSRead_ReadAds[udiActiveNumberOfSymbol_ReadAds].sFullSymbolName := Lynus_Standards.GVL_Communicator.arrInterfaceInfoAlVariables[byReadWriteArrayNumber,udiActiveNumberOfSymbol_ReadAds].sFullSymbolName;
							stADSRead_ReadAds[udiActiveNumberOfSymbol_ReadAds].arrValue := arrValueDefault_ReadAds;	
								IF Lynus_Standards.GVL_Communicator.arrInterfaceInfoAlVariables[byReadWriteArrayNumber,udiActiveNumberOfSymbol_ReadAds].uiSizeArray <= Lynus_Standards.Constants_Communicator.bySizeOfValueArray THEN  
									FOR uiLPWriteValueByArray_ReadAds := 1 TO Lynus_Standards.GVL_Communicator.arrInterfaceInfoAlVariables[byReadWriteArrayNumber,udiActiveNumberOfSymbol_ReadAds].uiSizeArray BY 1 DO
										arrCounterWriteValueInArray_ReadAds[1] := LIMIT(1,arrCounterWriteValueInArray_ReadAds[1],1600); arrCounterWriteValueInArray_ReadAds[2] := LIMIT(2,arrCounterWriteValueInArray_ReadAds[2],1600);
											arrCounterWriteValueInArray_ReadAds[3] := LIMIT(3,arrCounterWriteValueInArray_ReadAds[3],1600); arrCounterWriteValueInArray_ReadAds[4] := LIMIT(4,arrCounterWriteValueInArray_ReadAds[4],1600);
												arrCounterWriteValueInArray_ReadAds[5] := LIMIT(5,arrCounterWriteValueInArray_ReadAds[5],1600); arrCounterWriteValueInArray_ReadAds[6] := LIMIT(6,arrCounterWriteValueInArray_ReadAds[6],1600);
													arrCounterWriteValueInArray_ReadAds[7] := LIMIT(7,arrCounterWriteValueInArray_ReadAds[7],1600); arrCounterWriteValueInArray_ReadAds[8] := LIMIT(8,arrCounterWriteValueInArray_ReadAds[8],1600);
														unConvertULINT_TO_LREAL_ReadAds.uliRawValue := LINT_TO_ULINT(ULINT_TO_LINT(SHL(BYTE_TO_ULINT(arrValueAfterRead_ReadAds[arrCounterWriteValueInArray_ReadAds[8]]),56) + SHL(BYTE_TO_ULINT(arrValueAfterRead_ReadAds[arrCounterWriteValueInArray_ReadAds[7]]),48) + SHL(BYTE_TO_ULINT(arrValueAfterRead_ReadAds[arrCounterWriteValueInArray_ReadAds[6]]),40) + SHL(BYTE_TO_ULINT(arrValueAfterRead_ReadAds[arrCounterWriteValueInArray_ReadAds[5]]),32) +
																											SHL(BYTE_TO_ULINT(arrValueAfterRead_ReadAds[arrCounterWriteValueInArray_ReadAds[4]]),24) + SHL(BYTE_TO_ULINT(arrValueAfterRead_ReadAds[arrCounterWriteValueInArray_ReadAds[3]]),16) + SHL(BYTE_TO_ULINT(arrValueAfterRead_ReadAds[arrCounterWriteValueInArray_ReadAds[2]]),8) + BYTE_TO_ULINT(arrValueAfterRead_ReadAds[arrCounterWriteValueInArray_ReadAds[1]])));
										arrCounterWriteValueInArray_ReadAds[1] := arrCounterWriteValueInArray_ReadAds[1] + 8; arrCounterWriteValueInArray_ReadAds[2] := arrCounterWriteValueInArray_ReadAds[2] + 8;
											arrCounterWriteValueInArray_ReadAds[3] := arrCounterWriteValueInArray_ReadAds[3] + 8; arrCounterWriteValueInArray_ReadAds[4] := arrCounterWriteValueInArray_ReadAds[4] + 8;
												arrCounterWriteValueInArray_ReadAds[5] := arrCounterWriteValueInArray_ReadAds[5] + 8; arrCounterWriteValueInArray_ReadAds[6] := arrCounterWriteValueInArray_ReadAds[6] + 8;
													arrCounterWriteValueInArray_ReadAds[7] := arrCounterWriteValueInArray_ReadAds[7] + 8; arrCounterWriteValueInArray_ReadAds[8] := arrCounterWriteValueInArray_ReadAds[8] + 8;			
														IF IsFinite(F_LREAL(unConvertULINT_TO_LREAL_ReadAds.lrValueFloat)) THEN
															IF LEN(LREAL_TO_STRING(unConvertULINT_TO_LREAL_ReadAds.lrValueFloat)) <= 30 THEN 
																IF FIND(LREAL_TO_STRING(unConvertULINT_TO_LREAL_ReadAds.lrValueFloat),'e') = 0 AND FIND(LREAL_TO_STRING(unConvertULINT_TO_LREAL_ReadAds.lrValueFloat),'E') = 0 THEN 
																	sStringFloat_ReadAds := LREAL_TO_STRING(unConvertULINT_TO_LREAL_ReadAds.lrValueFloat);
																		iFindPointFloat_ReadAds := FIND(sStringFloat_ReadAds,'.');
																			sStringFloat_ReadAds := DELETE(sStringFloat_ReadAds,iFindPointFloat_ReadAds,1);
																				iPrecision_ReadAds := LEN(sStringFloat_ReadAds);
																					iPrecision_ReadAds := LIMIT(0,iPrecision_ReadAds,16);
																	IF LEN(LREAL_TO_FMTSTR(unConvertULINT_TO_LREAL_ReadAds.lrValueFloat,iPrecision_ReadAds,TRUE)) <= 30 THEN
																		//Check if the output from Function LREAL_TO_FMTSTR is ok 
																		IF LREAL_TO_FMTSTR(unConvertULINT_TO_LREAL_ReadAds.lrValueFloat,iPrecision_ReadAds,TRUE) <> '#INF' AND LREAL_TO_FMTSTR(unConvertULINT_TO_LREAL_ReadAds.lrValueFloat,iPrecision_ReadAds,TRUE) <> '-#INF' AND
																			LREAL_TO_FMTSTR(unConvertULINT_TO_LREAL_ReadAds.lrValueFloat,iPrecision_ReadAds,TRUE) <> '#QNAN' AND LREAL_TO_FMTSTR(unConvertULINT_TO_LREAL_ReadAds.lrValueFloat,iPrecision_ReadAds,TRUE) <> '-#QNAN' AND
																				LREAL_TO_FMTSTR(unConvertULINT_TO_LREAL_ReadAds.lrValueFloat,iPrecision_ReadAds,TRUE) <> '#OVF' AND LREAL_TO_FMTSTR(unConvertULINT_TO_LREAL_ReadAds.lrValueFloat,iPrecision_ReadAds,TRUE) <> '-#OVF' THEN
																					stADSRead_ReadAds[udiActiveNumberOfSymbol_ReadAds].arrValue[uiLPWriteValueByArray_ReadAds] := LREAL_TO_FMTSTR(unConvertULINT_TO_LREAL_ReadAds.lrValueFloat,iPrecision_ReadAds,TRUE); 
																		ELSE
																			iState_ReadAds := 200;
																				uiInternError_ReadAds := 1;
																		END_IF
																	ELSE
																		//Check if the output from Function LREAL_TO_FMTSTR is ok 
																		IF MID(LREAL_TO_FMTSTR(unConvertULINT_TO_LREAL_ReadAds.lrValueFloat,iPrecision_ReadAds,TRUE),30,1) <> '#INF' AND MID(LREAL_TO_FMTSTR(unConvertULINT_TO_LREAL_ReadAds.lrValueFloat,iPrecision_ReadAds,TRUE),30,1) <> '-#INF' AND
																			MID(LREAL_TO_FMTSTR(unConvertULINT_TO_LREAL_ReadAds.lrValueFloat,iPrecision_ReadAds,TRUE),30,1) <> '#QNAN' AND MID(LREAL_TO_FMTSTR(unConvertULINT_TO_LREAL_ReadAds.lrValueFloat,iPrecision_ReadAds,TRUE),30,1) <> '-#QNAN' AND
																				MID(LREAL_TO_FMTSTR(unConvertULINT_TO_LREAL_ReadAds.lrValueFloat,iPrecision_ReadAds,TRUE),30,1) <> '#OVF' AND MID(LREAL_TO_FMTSTR(unConvertULINT_TO_LREAL_ReadAds.lrValueFloat,iPrecision_ReadAds,TRUE),30,1) <> '-#OVF' THEN
																					stADSRead_ReadAds[udiActiveNumberOfSymbol_ReadAds].arrValue[uiLPWriteValueByArray_ReadAds] := MID(LREAL_TO_FMTSTR(unConvertULINT_TO_LREAL_ReadAds.lrValueFloat,iPrecision_ReadAds,TRUE),30,1);
																		ELSE
																			iState_ReadAds := 200;
																				uiInternError_ReadAds := 1;
																		END_IF 
																	END_IF
																ELSE
																	stADSRead_ReadAds[udiActiveNumberOfSymbol_ReadAds].arrValue[uiLPWriteValueByArray_ReadAds] := LREAL_TO_STRING(unConvertULINT_TO_LREAL_ReadAds.lrValueFloat);
																END_IF
															ELSE
																iState_ReadAds := 200;
																	uiInternError_ReadAds := 1;
															END_IF
														ELSE
															iState_ReadAds := 200;
																uiInternError_ReadAds := 1;
														END_IF
									END_FOR 
								END_IF
					END_IF
				//ARRAY OF STRING(30)
				IF FIND(Lynus_Standards.GVL_Communicator.arrInterfaceInfoAlVariables[byReadWriteArrayNumber,udiActiveNumberOfSymbol_ReadAds].sSymbolType,'OF STRING(30)') <> 0 THEN
					stADSRead_ReadAds[udiActiveNumberOfSymbol_ReadAds].sFullSymbolName := Lynus_Standards.GVL_Communicator.arrInterfaceInfoAlVariables[byReadWriteArrayNumber,udiActiveNumberOfSymbol_ReadAds].sFullSymbolName;
						stADSRead_ReadAds[udiActiveNumberOfSymbol_ReadAds].arrValue := arrValueDefault_ReadAds;	
							IF Lynus_Standards.GVL_Communicator.arrInterfaceInfoAlVariables[byReadWriteArrayNumber,udiActiveNumberOfSymbol_ReadAds].uiSizeArray <= Lynus_Standards.Constants_Communicator.bySizeOfValueArray THEN
								FOR uiLPWriteValueByArray_ReadAds := 1 TO Lynus_Standards.Constants_Communicator.bySizeOfValueArray BY 1 DO 
									FOR byLPCheckCharactersAfterReadOut_ReadAds := 1 TO 31 BY 1 DO
										uiCounterArrayOfString_ReadAds := uiCounterArrayOfString_ReadAds + 1;
											uiCounterArrayOfString_ReadAds := LIMIT(1,uiCounterArrayOfString_ReadAds,1600);	
												stADSRead_ReadAds[udiActiveNumberOfSymbol_ReadAds].arrValue[uiLPWriteValueByArray_ReadAds] := CONCAT(stADSRead_ReadAds[udiActiveNumberOfSymbol_ReadAds].arrValue[uiLPWriteValueByArray_ReadAds],F_ToCHR(arrValueAfterRead_ReadAds[uiCounterArrayOfString_ReadAds]));
													IF arrValueAfterRead_ReadAds[uiCounterArrayOfString_ReadAds] = 0 AND stADSRead_ReadAds[udiActiveNumberOfSymbol_ReadAds].arrValue[uiLPWriteValueByArray_ReadAds] <> '' THEN	
														uiCounterArrayOfString_ReadAds := 31 * uiLPWriteValueByArray_ReadAds;	    
															EXIT; 
													ELSIF arrValueAfterRead_ReadAds[uiCounterArrayOfString_ReadAds] = 0 AND stADSRead_ReadAds[udiActiveNumberOfSymbol_ReadAds].arrValue[uiLPWriteValueByArray_ReadAds] = '' THEN 
														stADSRead_ReadAds[udiActiveNumberOfSymbol_ReadAds].arrValue[uiLPWriteValueByArray_ReadAds] := '#EMPTY#';
															uiCounterArrayOfString_ReadAds := 31 * uiLPWriteValueByArray_ReadAds;
																EXIT;	
													END_IF 
									END_FOR
								END_FOR 
				END_IF		END_IF
					//ARRAY OF TIME or ARRAY OF TIME OF DAY	
					IF FIND(Lynus_Standards.GVL_Communicator.arrInterfaceInfoAlVariables[byReadWriteArrayNumber,udiActiveNumberOfSymbol_ReadAds].sSymbolType,'OF TIME') <> 0 OR FIND(Lynus_Standards.GVL_Communicator.arrInterfaceInfoAlVariables[byReadWriteArrayNumber,udiActiveNumberOfSymbol_ReadAds].sSymbolType,'OF TIME_OF_DAY') <> 0 THEN
						stADSRead_ReadAds[udiActiveNumberOfSymbol_ReadAds].sFullSymbolName := Lynus_Standards.GVL_Communicator.arrInterfaceInfoAlVariables[byReadWriteArrayNumber,udiActiveNumberOfSymbol_ReadAds].sFullSymbolName;
							stADSRead_ReadAds[udiActiveNumberOfSymbol_ReadAds].arrValue := arrValueDefault_ReadAds;	
								IF Lynus_Standards.GVL_Communicator.arrInterfaceInfoAlVariables[byReadWriteArrayNumber,udiActiveNumberOfSymbol_ReadAds].uiSizeArray <= Lynus_Standards.Constants_Communicator.bySizeOfValueArray THEN  
									FOR uiLPWriteValueByArray_ReadAds := 1 TO Lynus_Standards.GVL_Communicator.arrInterfaceInfoAlVariables[byReadWriteArrayNumber,udiActiveNumberOfSymbol_ReadAds].uiSizeArray BY 1 DO
										arrCounterWriteValueInArray_ReadAds[1] := LIMIT(1,arrCounterWriteValueInArray_ReadAds[1],1600); arrCounterWriteValueInArray_ReadAds[2] := LIMIT(2,arrCounterWriteValueInArray_ReadAds[2],1600);
											arrCounterWriteValueInArray_ReadAds[3] := LIMIT(3,arrCounterWriteValueInArray_ReadAds[3],1600); arrCounterWriteValueInArray_ReadAds[4] := LIMIT(4,arrCounterWriteValueInArray_ReadAds[4],1600);
												stADSRead_ReadAds[udiActiveNumberOfSymbol_ReadAds].arrValue[uiLPWriteValueByArray_ReadAds] := UDINT_TO_STRING(SHL(BYTE_TO_UDINT(arrValueAfterRead_ReadAds[arrCounterWriteValueInArray_ReadAds[4]]),24) + SHL(BYTE_TO_UDINT(arrValueAfterRead_ReadAds[arrCounterWriteValueInArray_ReadAds[3]]),16) + SHL(BYTE_TO_UDINT(arrValueAfterRead_ReadAds[arrCounterWriteValueInArray_ReadAds[2]]),8) + BYTE_TO_UDINT(arrValueAfterRead_ReadAds[arrCounterWriteValueInArray_ReadAds[1]]));
										arrCounterWriteValueInArray_ReadAds[1] := arrCounterWriteValueInArray_ReadAds[1] + 4; arrCounterWriteValueInArray_ReadAds[2] := arrCounterWriteValueInArray_ReadAds[2] + 4;
											arrCounterWriteValueInArray_ReadAds[3] := arrCounterWriteValueInArray_ReadAds[3] + 4; arrCounterWriteValueInArray_ReadAds[4] := arrCounterWriteValueInArray_ReadAds[4] + 4;
									END_FOR 
								END_IF
					END_IF
				//ARRAY OF DATE or ARRAY OF DATE AND TIME
				IF FIND(Lynus_Standards.GVL_Communicator.arrInterfaceInfoAlVariables[byReadWriteArrayNumber,udiActiveNumberOfSymbol_ReadAds].sSymbolType,'OF DATE') <> 0 OR FIND(Lynus_Standards.GVL_Communicator.arrInterfaceInfoAlVariables[byReadWriteArrayNumber,udiActiveNumberOfSymbol_ReadAds].sSymbolType,'OF DATE_AND_TIME') <> 0 THEN
					stADSRead_ReadAds[udiActiveNumberOfSymbol_ReadAds].sFullSymbolName := Lynus_Standards.GVL_Communicator.arrInterfaceInfoAlVariables[byReadWriteArrayNumber,udiActiveNumberOfSymbol_ReadAds].sFullSymbolName;
						stADSRead_ReadAds[udiActiveNumberOfSymbol_ReadAds].arrValue := arrValueDefault_ReadAds;	
							IF Lynus_Standards.GVL_Communicator.arrInterfaceInfoAlVariables[byReadWriteArrayNumber,udiActiveNumberOfSymbol_ReadAds].uiSizeArray <= Lynus_Standards.Constants_Communicator.bySizeOfValueArray THEN  
								FOR uiLPWriteValueByArray_ReadAds := 1 TO Lynus_Standards.GVL_Communicator.arrInterfaceInfoAlVariables[byReadWriteArrayNumber,udiActiveNumberOfSymbol_ReadAds].uiSizeArray BY 1 DO
									arrCounterWriteValueInArray_ReadAds[1] := LIMIT(1,arrCounterWriteValueInArray_ReadAds[1],1600); arrCounterWriteValueInArray_ReadAds[2] := LIMIT(2,arrCounterWriteValueInArray_ReadAds[2],1600);
										arrCounterWriteValueInArray_ReadAds[3] := LIMIT(3,arrCounterWriteValueInArray_ReadAds[3],1600); arrCounterWriteValueInArray_ReadAds[4] := LIMIT(4,arrCounterWriteValueInArray_ReadAds[4],1600);
											uliValueDateTime_ReadAds := SHL(BYTE_TO_UDINT(arrValueAfterRead_ReadAds[arrCounterWriteValueInArray_ReadAds[4]]),24) + SHL(BYTE_TO_UDINT(arrValueAfterRead_ReadAds[arrCounterWriteValueInArray_ReadAds[3]]),16) + SHL(BYTE_TO_UDINT(arrValueAfterRead_ReadAds[arrCounterWriteValueInArray_ReadAds[2]]),8) + BYTE_TO_UDINT(arrValueAfterRead_ReadAds[arrCounterWriteValueInArray_ReadAds[1]]);
												uliValueDateTime_ReadAds := uliValueDateTime_ReadAds * 1000;	
													stADSRead_ReadAds[udiActiveNumberOfSymbol_ReadAds].arrValue[uiLPWriteValueByArray_ReadAds] := ULINT_TO_STRING(uliValueDateTime_ReadAds); 
									arrCounterWriteValueInArray_ReadAds[1] := arrCounterWriteValueInArray_ReadAds[1] + 4; arrCounterWriteValueInArray_ReadAds[2] := arrCounterWriteValueInArray_ReadAds[2] + 4;
										arrCounterWriteValueInArray_ReadAds[3] := arrCounterWriteValueInArray_ReadAds[3] + 4; arrCounterWriteValueInArray_ReadAds[4] := arrCounterWriteValueInArray_ReadAds[4] + 4;
								END_FOR 
							END_IF
				END_IF
					
			IF Lynus_Standards.GVL_Communicator.arrInterfaceInfoAlVariables[byReadWriteArrayNumber,udiActiveNumberOfSymbol_ReadAds].uiSizeArray <= Lynus_Standards.Constants_Communicator.bySizeOfValueArray AND iState_ReadAds = 5 THEN 
				arrCounterWriteValueInArray_ReadAds[1] := 0; arrCounterWriteValueInArray_ReadAds[2] := 0; arrCounterWriteValueInArray_ReadAds[3] := 0; 
				arrCounterWriteValueInArray_ReadAds[4] := 0; arrCounterWriteValueInArray_ReadAds[5] := 0; arrCounterWriteValueInArray_ReadAds[6] := 0; 
				arrCounterWriteValueInArray_ReadAds[7] := 0; arrCounterWriteValueInArray_ReadAds[8] := 0;
				uiCounterArrayOfString_ReadAds := 0;
				sStringFloat_ReadAds := ''; iFindPointFloat_ReadAds := 0; iPrecision_ReadAds := 0;
				iState_ReadAds := 6;
			 END_IF			
			
			IF timTimout_ReadAds.Q THEN iState_ReadAds := 200; END_IF
		
		ELSE
			IF udiActiveNumberOfSymbol_ReadAds < Lynus_Standards.GVL_Communicator.arrCounterVariableInArray[byReadWriteArrayNumber] AND udiNumberInProgress_ReadAds < udiNumberSizeValues_ReadAds THEN iState_ReadAds := -4; udiNumberInProgress_ReadAds := udiNumberInProgress_ReadAds + 1; END_IF
			IF (udiNumberInProgress_ReadAds >= udiNumberSizeValues_ReadAds AND iState_ReadAds = 5) THEN iState_ReadAds := -8; udiNumberInProgress_ReadAds := 0; END_IF
			IF udiActiveNumberOfSymbol_ReadAds >= Lynus_Standards.GVL_Communicator.arrCounterVariableInArray[byReadWriteArrayNumber] THEN iState_ReadAds := -8; udiActiveNumberOfSymbol_ReadAds := 0; udiNumberInProgress_ReadAds := 0; udiRestValueSymbolRead_ReadAds := 0; END_IF 
				//Timeout
				IF timTimout_ReadAds.Q THEN iState_ReadAds := 200; END_IF
		END_IF
	
	6://Check if the symbol exist
		byCounterWaitInStep_ReadAds := byCounterWaitInStep_ReadAds + 1;
			byCounterWaitInStep_ReadAds := LIMIT(1,byCounterWaitInStep_ReadAds,2);	
	
		IF byCounterWaitInStep_ReadAds = 1 THEN
			FOR udiLPCheckReadArrays_ReadAds := 1 TO udiNumberLoopHalf_ReadAds BY 1 DO
				IF stADSReadNew_ReadAds[udiLPCheckReadArrays_ReadAds].sFullSymbolName = Lynus_Standards.GVL_Communicator.arrInterfaceInfoAlVariables[byReadWriteArrayNumber,udiActiveNumberOfSymbol_ReadAds].sFullSymbolName THEN 
					iState_ReadAds := 7;																				//Symbol exist in the read array
				END_IF
			END_FOR
		END_IF
			IF byCounterWaitInStep_ReadAds = 2 AND udiNumberLoopFull_ReadAds <> udiNumberLoopHalf_ReadAds THEN
				FOR udiLPCheckReadArrays_ReadAds := (udiNumberLoopHalf_ReadAds + 1) TO udiNumberLoopFull_ReadAds BY 1 DO
					IF stADSReadNew_ReadAds[udiLPCheckReadArrays_ReadAds].sFullSymbolName = Lynus_Standards.GVL_Communicator.arrInterfaceInfoAlVariables[byReadWriteArrayNumber,udiActiveNumberOfSymbol_ReadAds].sFullSymbolName THEN 
						iState_ReadAds := 7;																			//Symbol exist in the read array
					END_IF
				END_FOR
			END_IF
		
				IF byCounterWaitInStep_ReadAds >= 2 AND iState_ReadAds = 6 THEN iState_ReadAds := 9; END_IF 			//Symbol not exist	
				
			//Timeout
			IF timTimout_ReadAds.Q THEN iState_ReadAds := 200; END_IF		
				
	7://Check if the value has changed
		byCounterWaitInStep_ReadAds := 0;
			bValueIsTheSame_ReadAds := FALSE;	
		
		FOR byLPCheckValueChange_ReadAds := 1 TO Lynus_Standards.Constants_Communicator.bySizeOfValueArray BY 1 DO
			IF (stADSRead_ReadAds[udiActiveNumberOfSymbol_ReadAds].arrValue[byLPCheckValueChange_ReadAds] <> stADSReadNew_ReadAds[udiActiveNumberOfSymbol_ReadAds].arrValue[byLPCheckValueChange_ReadAds] AND m_EnableChange_upload)    // Stefan added AND 
			OR m_TriggerIntervalSend THEN		// Stefan
				iState_ReadAds := 8;																																				//Value has changed
			ELSE		
				IF iState_ReadAds = 7 AND byLPCheckValueChange_ReadAds >= Lynus_Standards.Constants_Communicator.bySizeOfValueArray THEN iState_ReadAds := 10; bValueIsTheSame_ReadAds := TRUE; END_IF		//Value is the same
			END_IF 
		END_FOR	
		
			//Timeout
			IF timTimout_ReadAds.Q THEN iState_ReadAds := 200; END_IF	
		
	8://Symbol exist and Value has changed
		byCounterWaitInStep_ReadAds := byCounterWaitInStep_ReadAds + 1;
			byCounterWaitInStep_ReadAds := LIMIT(1,byCounterWaitInStep_ReadAds,2);
	
		IF byCounterWaitInStep_ReadAds = 1 THEN 
			FOR udiLPCheckReadArrays_ReadAds := 1 TO udiNumberLoopHalf_ReadAds BY 1 DO
				IF stADSRead_ReadAds[udiLPCheckReadArrays_ReadAds].sFullSymbolName = stADSReadNew_ReadAds[udiLPCheckReadArrays_ReadAds].sFullSymbolName THEN
					stADSReadNew_ReadAds[udiLPCheckReadArrays_ReadAds].arrValue := stADSRead_ReadAds[udiLPCheckReadArrays_ReadAds].arrValue;
				END_IF
			END_FOR
		END_IF	
			IF byCounterWaitInStep_ReadAds = 2 AND udiNumberLoopFull_ReadAds <> udiNumberLoopHalf_ReadAds THEN 
				FOR udiLPCheckReadArrays_ReadAds := (udiNumberLoopHalf_ReadAds + 1) TO udiNumberLoopFull_ReadAds BY 1 DO
					IF stADSRead_ReadAds[udiLPCheckReadArrays_ReadAds].sFullSymbolName = stADSReadNew_ReadAds[udiLPCheckReadArrays_ReadAds].sFullSymbolName THEN
						stADSReadNew_ReadAds[udiLPCheckReadArrays_ReadAds].arrValue := stADSRead_ReadAds[udiLPCheckReadArrays_ReadAds].arrValue;	
					END_IF
				END_FOR
			END_IF 
		
				IF byCounterWaitInStep_ReadAds >= 2 THEN iState_ReadAds := 10; END_IF			
		
			//Timeout
			IF timTimout_ReadAds.Q THEN iState_ReadAds := 200; END_IF
		
	9://Copy the new symbol in the array
		byCounterWaitInStep_ReadAds := 0;
			stADSReadNew_ReadAds := stADSRead_ReadAds;
				iState_ReadAds := 10;
			
	10://Write in Buffer if the send bus is busy or send a messege if the buffer is not empty
		byCounterWaitInStep_ReadAds := 0;
	
		IF NOT Lynus_Standards.GVL_Communicator.arrInterfaceInfoValueSendTo[byReadWriteArrayNumber].bBusy THEN	
			Lynus_Standards.GVL_Communicator.arrInterfaceInfoValueSendTo[byReadWriteArrayNumber].arrValue := arrValueDefault_ReadAds; 						//Clear send Interface if it is no message to send
				Lynus_Standards.GVL_Communicator.arrInterfaceInfoValueSendTo[byReadWriteArrayNumber].sSymbolUnit := ''; 
					Lynus_Standards.GVL_Communicator.arrInterfaceInfoValueSendTo[byReadWriteArrayNumber].sFullSymbolName := '';
						Lynus_Standards.GVL_Communicator.arrInterfaceInfoValueSendTo[byReadWriteArrayNumber].sSymbolType := '';
							IF fbBuffer_ReadAds.nCount > 0 THEN							
								iState_ReadAds := 11;														//Send a new messege from the buffer
							END_IF																			
		END_IF
			IF ((Lynus_Standards.GVL_Communicator.arrInterfaceInfoValueSendTo[byReadWriteArrayNumber].bBusy OR fbBuffer_ReadAds.nCount = 0) AND NOT bValueIsTheSame_ReadAds) THEN
				iState_ReadAds := 20;																		//Insert a new value in the buffer if the send bus is busy or no value is stored in the buffer
			ELSE
				IF iState_ReadAds = 10 THEN 																						
					iState_ReadAds := 100;																	//Value is the same
				END_IF																						
			END_IF
		
			//Timeout
			IF timTimout_ReadAds.Q THEN iState_ReadAds := 200; END_IF
	
	11://Read out a Value from the buffer for sending
		IF udiCounterReadBuffer_New_ReadAds <> fbBuffer_ReadAds.nCount AND fbBuffer_ReadAds.bOk THEN
			udiCounterReadBuffer_New_ReadAds := fbBuffer_ReadAds.nCount;
				IF fbBuffer_ReadAds.cbReturn <= 2000 THEN 
					FOR udiLPCheckReadBuffer_ReadAds := 1 TO fbBuffer_ReadAds.cbReturn BY 1 DO	
						IF byCounterValueReadOut_ReadAds = 0 AND arrBufferRead_ReadAds[udiLPCheckReadBuffer_ReadAds] <> 59 THEN sSymbolNameOutFromBuffer_ReadAds := CONCAT(sSymbolNameOutFromBuffer_ReadAds,F_ToCHR(arrBufferRead_ReadAds[udiLPCheckReadBuffer_ReadAds])); END_IF 
							IF arrBufferRead_ReadAds[udiLPCheckReadBuffer_ReadAds] = 59 THEN byCounterValueReadOut_ReadAds := byCounterValueReadOut_ReadAds + 1; END_IF
								byCounterValueReadOut_ReadAds := LIMIT(0,byCounterValueReadOut_ReadAds,Lynus_Standards.Constants_Communicator.bySizeOfValueArray);
									IF byCounterValueReadOut_ReadAds >= 1 AND arrBufferRead_ReadAds[udiLPCheckReadBuffer_ReadAds] <> 59 AND arrBufferRead_ReadAds[udiLPCheckReadBuffer_ReadAds] <> 0 THEN 
										arrValueOutFromBuffer_ReadAds[byCounterValueReadOut_ReadAds] := CONCAT(arrValueOutFromBuffer_ReadAds[byCounterValueReadOut_ReadAds],F_ToCHR(arrBufferRead_ReadAds[udiLPCheckReadBuffer_ReadAds])); 
									END_IF    	
					END_FOR				 
						IF arrBufferRead_ReadAds[udiLPCheckReadBuffer_ReadAds] = 0 THEN iState_ReadAds := 12; byCounterValueReadOut_ReadAds := 0; END_IF
				END_IF
		END_IF
		
			IF timTimout_ReadAds.Q THEN iState_ReadAds := 200; END_IF
	
	12://Write the Date on interface and start the sending
		byCounterWaitInStep_ReadAds := byCounterWaitInStep_ReadAds + 1;
			byCounterWaitInStep_ReadAds := LIMIT(1,byCounterWaitInStep_ReadAds,2);
	
		IF byCounterWaitInStep_ReadAds = 1 THEN 
			FOR udiLPCheckVarInfoBeforSending_ReadAds := 1 TO udiNumberLoopHalf_ReadAds BY 1 DO
				IF Lynus_Standards.GVL_Communicator.arrInterfaceInfoAlVariables[byReadWriteArrayNumber,udiLPCheckVarInfoBeforSending_ReadAds].sFullSymbolName = sSymbolNameOutFromBuffer_ReadAds THEN
					Lynus_Standards.GVL_Communicator.arrInterfaceInfoValueSendTo[byReadWriteArrayNumber].sFullSymbolName := sSymbolNameOutFromBuffer_ReadAds;
						Lynus_Standards.GVL_Communicator.arrInterfaceInfoValueSendTo[byReadWriteArrayNumber].sSymbolUnit := Lynus_Standards.GVL_Communicator.arrInterfaceInfoAlVariables[byReadWriteArrayNumber,udiLPCheckVarInfoBeforSending_ReadAds].sSymbolUnit;
							Lynus_Standards.GVL_Communicator.arrInterfaceInfoValueSendTo[byReadWriteArrayNumber].sSymbolType := Lynus_Standards.GVL_Communicator.arrInterfaceInfoAlVariables[byReadWriteArrayNumber,udiLPCheckVarInfoBeforSending_ReadAds].sSymbolType;
								Lynus_Standards.GVL_Communicator.arrInterfaceInfoValueSendTo[byReadWriteArrayNumber].arrValue := arrValueOutFromBuffer_ReadAds;
									Lynus_Standards.GVL_Communicator.arrInterfaceInfoValueSendTo[byReadWriteArrayNumber].bBusy := TRUE;
										iState_ReadAds := 13;
											EXIT;	
				END_IF 		 	   	
			END_FOR 	
		END_IF
			IF byCounterWaitInStep_ReadAds = 2 AND udiNumberLoopFull_ReadAds <> udiNumberLoopHalf_ReadAds THEN 
				FOR udiLPCheckVarInfoBeforSending_ReadAds := (udiNumberLoopHalf_ReadAds + 1) TO udiNumberLoopFull_ReadAds BY 1 DO
					IF Lynus_Standards.GVL_Communicator.arrInterfaceInfoAlVariables[byReadWriteArrayNumber,udiLPCheckVarInfoBeforSending_ReadAds].sFullSymbolName = sSymbolNameOutFromBuffer_ReadAds THEN
						Lynus_Standards.GVL_Communicator.arrInterfaceInfoValueSendTo[byReadWriteArrayNumber].sFullSymbolName := sSymbolNameOutFromBuffer_ReadAds;
							Lynus_Standards.GVL_Communicator.arrInterfaceInfoValueSendTo[byReadWriteArrayNumber].sSymbolUnit := Lynus_Standards.GVL_Communicator.arrInterfaceInfoAlVariables[byReadWriteArrayNumber,udiLPCheckVarInfoBeforSending_ReadAds].sSymbolUnit;
								Lynus_Standards.GVL_Communicator.arrInterfaceInfoValueSendTo[byReadWriteArrayNumber].sSymbolType := Lynus_Standards.GVL_Communicator.arrInterfaceInfoAlVariables[byReadWriteArrayNumber,udiLPCheckVarInfoBeforSending_ReadAds].sSymbolType;
									Lynus_Standards.GVL_Communicator.arrInterfaceInfoValueSendTo[byReadWriteArrayNumber].arrValue := arrValueOutFromBuffer_ReadAds;
										Lynus_Standards.GVL_Communicator.arrInterfaceInfoValueSendTo[byReadWriteArrayNumber].bBusy := TRUE;
											iState_ReadAds := 13;
												EXIT;	
					END_IF 		 	   	
				END_FOR 	
			END_IF
		
			IF timTimout_ReadAds.Q THEN iState_ReadAds := 200; END_IF
			
	13://Clear Read Buffer (conserve resources because the code must also work for small plc's)
		byCounterWaitInStep_ReadAds := 0;
			sSymbolNameOutFromBuffer_ReadAds := '';
				MEMCPY(ADR(arrBufferRead_ReadAds),ADR(arrBufferWriteReadDefault_ReadAds),SIZEOF(arrBufferRead_ReadAds));
					arrValueOutFromBuffer_ReadAds := arrValueDefault_ReadAds;
		
			iState_ReadAds := 10;
			
	20://Dim size from the values and symbol name befor can saving in buffer
		uiNumberValueSymbolSize_ReadAds := 0;
			byNumberOfValues_ReadAds_ReadAds := 0;
				byLenghSymbolName_ReadAds := 0;
		FOR byLPDimValueNumberASize_ReadAds := 1 TO Lynus_Standards.Constants_Communicator.bySizeOfValueArray BY 1 DO
			uiNumberValueSymbolSize_ReadAds := uiNumberValueSymbolSize_ReadAds + INT_TO_UINT(LEN(stADSReadNew_ReadAds[udiActiveNumberOfSymbol_ReadAds].arrValue[byLPDimValueNumberASize_ReadAds]));
				IF stADSReadNew_ReadAds[udiActiveNumberOfSymbol_ReadAds].arrValue[byLPDimValueNumberASize_ReadAds] <> '' THEN uiNumberValueSymbolSize_ReadAds := uiNumberValueSymbolSize_ReadAds + 1; END_IF 	
					IF stADSReadNew_ReadAds[udiActiveNumberOfSymbol_ReadAds].arrValue[byLPDimValueNumberASize_ReadAds] <> '' THEN byNumberOfValues_ReadAds_ReadAds := byNumberOfValues_ReadAds_ReadAds + 1; END_IF	
		END_FOR 	
			byLenghSymbolName_ReadAds := INT_TO_BYTE(LEN(stADSReadNew_ReadAds[udiActiveNumberOfSymbol_ReadAds].sFullSymbolName));
				uiNumberValueSymbolSize_ReadAds := uiNumberValueSymbolSize_ReadAds + byLenghSymbolName_ReadAds + 1;
		
			IF byNumberOfValues_ReadAds_ReadAds <= Lynus_Standards.Constants_Communicator.bySizeOfValueArray THEN
				FOR byLPDimLenghValues_ReadAds := 1 TO byNumberOfValues_ReadAds_ReadAds BY 1 DO
					arrLenghEachValue_ReadAds[byLPDimLenghValues_ReadAds] := INT_TO_BYTE(LEN(stADSReadNew_ReadAds[udiActiveNumberOfSymbol_ReadAds].arrValue[byLPDimLenghValues_ReadAds]));	
				END_FOR 
			END_IF
	
		IF byNumberOfValues_ReadAds_ReadAds <= Lynus_Standards.Constants_Communicator.bySizeOfValueArray AND byNumberOfValues_ReadAds_ReadAds >= 1 AND uiNumberValueSymbolSize_ReadAds <> 0 THEN iState_ReadAds := 21; END_IF
		
			IF timTimout_ReadAds.Q THEN iState_ReadAds := 200; END_IF
			
	21://String to Ascii Symbol Name and values
		IF byLenghSymbolName_ReadAds <= 49 THEN
			FOR byLPSymbolNameToAscii_ReadAds := 1 TO byLenghSymbolName_ReadAds BY 1 DO
				arrSymbolName_ReadAds[byLPSymbolNameToAscii_ReadAds] := F_ToASC(MID(stADSReadNew_ReadAds[udiActiveNumberOfSymbol_ReadAds].sFullSymbolName,1,byLPSymbolNameToAscii_ReadAds));
			END_FOR 
		END_IF
			IF byLenghSymbolName_ReadAds < 49 THEN arrSymbolName_ReadAds[byLenghSymbolName_ReadAds + 1] := F_ToASC(';'); END_IF  	
		
		IF byNumberOfValues_ReadAds_ReadAds <= Lynus_Standards.Constants_Communicator.bySizeOfValueArray THEN 
			FOR byLPValueNameToAscii_1_ReadAds := 1 TO byNumberOfValues_ReadAds_ReadAds BY 1 DO
				IF arrLenghEachValue_ReadAds[byLPValueNameToAscii_1_ReadAds] <= 31 THEN 
					FOR byLPValueNameToAscii_2_ReadAds := 1 TO arrLenghEachValue_ReadAds[byLPValueNameToAscii_1_ReadAds] BY 1 DO
						arrValueName_ReadAds[byLPValueNameToAscii_1_ReadAds,byLPValueNameToAscii_2_ReadAds] := F_ToASC(MID(stADSReadNew_ReadAds[udiActiveNumberOfSymbol_ReadAds].arrValue[byLPValueNameToAscii_1_ReadAds],1,byLPValueNameToAscii_2_ReadAds));
					END_FOR
				END_IF
					arrValueName_ReadAds[byLPValueNameToAscii_1_ReadAds,byLPValueNameToAscii_2_ReadAds] := F_ToASC(';'); 			
			END_FOR 
		END_IF 
		
		IF byLenghSymbolName_ReadAds <= 49 AND byNumberOfValues_ReadAds_ReadAds <= Lynus_Standards.Constants_Communicator.bySizeOfValueArray AND arrLenghEachValue_ReadAds[byNumberOfValues_ReadAds_ReadAds] <= 31 THEN iState_ReadAds := 22; END_IF
		
			IF timTimout_ReadAds.Q THEN iState_ReadAds := 200; END_IF	
			
	22://Prepare Write array for Buffer
		IF byLenghSymbolName_ReadAds <= 48 THEN
			FOR uiLPWriteByteValueInArray_ReadAds := 1 TO (byLenghSymbolName_ReadAds + 1) BY 1 DO
				arrBufferWrite_ReadAds[uiLPWriteByteValueInArray_ReadAds] := arrSymbolName_ReadAds[uiLPWriteByteValueInArray_ReadAds];
			END_FOR 
		END_IF
		
		IF byLenghSymbolName_ReadAds <= 48 THEN	iState_ReadAds := 23; END_IF
			
			IF timTimout_ReadAds.Q THEN iState_ReadAds := 200; END_IF
	
	23://Prepare Write array for Buffer
		uiValueForLoopStart_ReadAds := uiLPWriteByteValueInArray_ReadAds;
			byValueInTurn_ReadAds := byValueInTurn_ReadAds + 1;
				byValueInTurn_ReadAds := LIMIT(1,byValueInTurn_ReadAds,Lynus_Standards.Constants_Communicator.bySizeOfValueArray);
					uiValueForLoopStop_ReadAds := arrLenghEachValue_ReadAds[byValueInTurn_ReadAds] + uiValueForLoopStart_ReadAds;
						byCounterValue_ReadAds := 0;
							
							IF uiValueForLoopStart_ReadAds >= 1 AND uiValueForLoopStart_ReadAds <= 2000 AND uiValueForLoopStop_ReadAds >= 1 AND uiValueForLoopStop_ReadAds <= 2000 THEN 
								FOR uiLPWriteByteValueInArray_ReadAds := uiValueForLoopStart_ReadAds TO uiValueForLoopStop_ReadAds BY 1 DO
									byCounterValue_ReadAds :=  byCounterValue_ReadAds + 1;
										byCounterValue_ReadAds := LIMIT(1,byCounterValue_ReadAds,31);	
											arrBufferWrite_ReadAds[uiLPWriteByteValueInArray_ReadAds] := arrValueName_ReadAds[byValueInTurn_ReadAds,byCounterValue_ReadAds];
								END_FOR 
							END_IF
		
		IF byValueInTurn_ReadAds >= byNumberOfValues_ReadAds_ReadAds AND uiValueForLoopStart_ReadAds >= 1 AND uiValueForLoopStart_ReadAds <= 2000 AND uiValueForLoopStop_ReadAds >= 1 AND uiValueForLoopStop_ReadAds <= 2000 THEN 
			iState_ReadAds := 24; 
				uiValueForLoopStart_ReadAds := 0;
					byValueInTurn_ReadAds := 0;
						uiValueForLoopStop_ReadAds := 0;
							byCounterValue_ReadAds := 0;			
		END_IF
			
			IF timTimout_ReadAds.Q THEN iState_ReadAds := 200; END_IF

	24://Write Value in Buffer
		iState_ReadAds := 25; 
				
	25://Check if the new value is stored in the buffer
		IF fbBuffer_ReadAds.bOk AND fbBuffer_ReadAds.nCount <> udiCounterReadBuffer_New_ReadAds THEN udiCounterReadBuffer_New_ReadAds := fbBuffer_ReadAds.nCount; iState_ReadAds := 26; END_IF  	
			
			IF timTimout_ReadAds.Q THEN iState_ReadAds := 200; END_IF
		
	26://Clear the Write Buffer (conserve resources because the code must also work for small plc's)
		MEMCPY(ADR(arrBufferWrite_ReadAds),ADR(arrBufferWriteReadDefault_ReadAds),SIZEOF(arrBufferWrite_ReadAds));
		
			iState_ReadAds := 100;

	100://Check for other variable
		//Next symbol
		IF udiActiveNumberOfSymbol_ReadAds < Lynus_Standards.GVL_Communicator.arrCounterVariableInArray[byReadWriteArrayNumber] AND udiNumberInProgress_ReadAds < udiNumberSizeValues_ReadAds THEN iState_ReadAds := -4; udiNumberInProgress_ReadAds := udiNumberInProgress_ReadAds + 1; END_IF
			//Start with the next 10 Variables
			IF (udiNumberInProgress_ReadAds >= udiNumberSizeValues_ReadAds AND iState_ReadAds = 100) THEN 
				iState_ReadAds := -8; 
					udiNumberInProgress_ReadAds := 0;
			END_IF	
				//Start from New with the first 10 Variables 	
				IF udiActiveNumberOfSymbol_ReadAds >= Lynus_Standards.GVL_Communicator.arrCounterVariableInArray[byReadWriteArrayNumber] THEN
					iState_ReadAds := -8; 
						udiActiveNumberOfSymbol_ReadAds := 0;
							udiNumberInProgress_ReadAds := 0;
								udiRestValueSymbolRead_ReadAds := 0;
						 			bFirstReadCycleDone_ReadAds := TRUE; 
				END_IF			
			
			bError_ReadAds := FALSE;
				uiInternError_ReadAds := 0;
			
			IF timTimout_ReadAds.Q THEN iState_ReadAds := 200; END_IF
				
	200://Error
		bError_ReadAds := TRUE; fbADSREADWRITE_ReadAds.WRTRD := FALSE; bValueIsTheSame_ReadAds := FALSE; 
			udiActiveNumberOfSymbol_ReadAds := 0; byCounterWaitInStep_ReadAds := 0; udiNumberInProgress_ReadAds := 0; udiRestValueSymbolRead_ReadAds := 0;
		
		//Clear the write Buffer befor go to step 0 (conserve resources because the code must also work for small plc's)
		MEMCPY(ADR(arrBufferWrite_ReadAds),ADR(arrBufferWriteReadDefault_ReadAds),SIZEOF(arrBufferWrite_ReadAds));
		
		//Clear the read Buffer befor go to step 0 (conserve resources because the code must also work for small plc's)
		sSymbolNameOutFromBuffer_ReadAds := '';
			MEMCPY(ADR(arrBufferRead_ReadAds),ADR(arrBufferWriteReadDefault_ReadAds),SIZEOF(arrBufferRead_ReadAds));
				arrValueOutFromBuffer_ReadAds := arrValueDefault_ReadAds;
			
		//Count up when an error has occurred
		byErrorCounter_ReadAds := byErrorCounter_ReadAds + 1;		
				
			iState_ReadAds := 300;
	
	300://Wait in Error and clear the rest from the read and write buffer (conserve resources because the code must also work for small plc's)
		byCounterWaitInStep_ReadAds := byCounterWaitInStep_ReadAds + 1;
	
			//Restart new from in Step -8. No Reset from the complete System
			IF byCounterWaitInStep_ReadAds > 10 AND byErrorCounter_ReadAds <= 10 THEN byCounterWaitInStep_ReadAds := 0; iState_ReadAds := -8; END_IF
				//Restart new from in Step -10. Reset from the complete System after to much Errors
				IF byCounterWaitInStep_ReadAds > 10 AND byErrorCounter_ReadAds > 10 THEN 
						byCounterWaitInStep_ReadAds := 0; 
							//Reset Read Steps and start from new
							iState_ReadAds := -10;
								//Reset Write Steps and start from new
								iState_WriteAds := -2;
									byErrorCounter_ReadAds := 0; 
				END_IF
	
END_CASE	

//Resetting the error counter after not being in the error step for 30 min
timResetErrorCounter_ReadAds(IN:= byErrorCounter_ReadAds <> 0, PT:= T#30M, Q=> , ET=> );
	IF timResetErrorCounter_ReadAds.Q THEN byErrorCounter_ReadAds := 0; END_IF 

//Read Out Variable by ADS
fbADSREADWRITE_ReadAds(
	NETID:= fbNedID.AddrString, 
	PORT:= uiPort, 
	IDXGRP:= 16#F080, 
	IDXOFFS:= udiNumberSizeValues_ReadAds, 
	WRITELEN:= , 
	READLEN:= udiSizeReq_ReadAds, 
	SRCADDR:= , 
	DESTADDR:= ADR(arrValueRead_ReadAds), 
	WRTRD:= , 
	TMOUT:= T#5S, 
	BUSY=> , 
	ERR=> , 
	ERRID=> );

FPErrorReadWrite_ReadAds(CLK:= fbADSREADWRITE_ReadAds.ERR, Q=> );	
	
//Buffer Read Value from ADS
FPWriteValueToBufferStep25_ReadAds(CLK:= iState_ReadAds = 24, Q=> );
FPReadValueToBufferStep11_ReadAds(CLK:= iState_ReadAds = 11, Q=> );

IF FPReadValueToBufferStep11_ReadAds.Q THEN fbBuffer_ReadAds.A_RemoveHead(); END_IF
IF FPWriteValueToBufferStep25_ReadAds.Q THEN fbBuffer_ReadAds.A_AddTail(); END_IF

//Reset the Buffer after a Buffer Overflow
IF fbBuffer_ReadAds.nCount <> 0 AND NOT fbBuffer_ReadAds.bOk THEN timResetBuffer_ReadAds.IN := TRUE; ELSE timResetBuffer_ReadAds.IN := FALSE; END_IF
	timResetBuffer_ReadAds(IN:= , PT:= T#40S, Q=> , ET=> );
		IF timResetBuffer_ReadAds.Q THEN fbBuffer_ReadAds.A_Reset(); END_IF

fbBuffer_ReadAds(
	pWrite:= ADR(arrBufferWrite_ReadAds), 
	cbWrite:= uiNumberValueSymbolSize_ReadAds, 
	pRead:= ADR(arrBufferRead_ReadAds), 
	cbRead:= SIZEOF(arrBufferRead_ReadAds), 
	pBuffer:= ADR(arrBufferADSRead_ReadAds), 
	cbBuffer:= SIZEOF(arrBufferADSRead_ReadAds), 
	bOk=> Lynus_Standards.GVL_Communicator.arrInterfaceInfoValueSendTo[byReadWriteArrayNumber].bBufferOK, 
	nCount=> Lynus_Standards.GVL_Communicator.arrInterfaceInfoValueSendTo[byReadWriteArrayNumber].udiCountBuffer, 
	cbSize=> , 
	cbReturn=> );

END_IF
	
//Busy
IF iState_ReadAds >= -8 OR iState_WriteAds >= 0 THEN bBusy := TRUE; ELSE bBusy := FALSE; END_IF
	
//Error
IF (bError_ReadAds AND iState_ReadAds <> - 10 AND iState_ReadAds <> - 9) OR (bError_WriteAds AND iState_WriteAds <> - 1 AND iState_WriteAds <> - 2) THEN fbErrorCodes.bErrorIntern := TRUE; ELSE fbErrorCodes.bErrorIntern := FALSE; END_IF

IF fbADSREADWRITE_ReadAds.ERR OR fbADSREADWRITE_WriteAds.ERR OR fbADSWrite_WriteAds.ERR THEN fbErrorCodes.bErrorADS := TRUE; END_IF

IF fbADSREADWRITE_ReadAds.ERR THEN fbErrorCodes.udiErrorCodeADS := fbADSREADWRITE_ReadAds.ERRID; END_IF
IF fbADSREADWRITE_WriteAds.ERR THEN fbErrorCodes.udiErrorCodeADS := fbADSREADWRITE_WriteAds.ERRID; END_IF
IF fbADSWrite_WriteAds.ERR THEN fbErrorCodes.udiErrorCodeADS := fbADSWrite_WriteAds.ERRID; END_IF

IF NOT fbADSREADWRITE_ReadAds.ERR AND NOT fbADSREADWRITE_ReadAds.BUSY AND NOT
	fbADSREADWRITE_WriteAds.ERR AND NOT fbADSREADWRITE_WriteAds.BUSY AND NOT fbADSWrite_WriteAds.ERR AND NOT fbADSWrite_WriteAds.BUSY THEN 
		fbErrorCodes.bErrorADS := FALSE;
			fbErrorCodes.udiErrorCodeADS := 0; 
END_IF 	     
	
fbErrorCodes(
	bErrorADS:= , 
	bErrorIntern:= , 
	udiErrorCodeADS:= , 
	udiErrorCodesInternRead:= uiInternError_ReadAds, 
	udiErrorCodesInternWrite:= uiInternError_WriteAds, 
	udiErrorCodeADS_Out=> udiErrorCodeOut, 
	bError=> bError, 
	eErrorReadWrite_Out=> eErrorReadWrite_Out);
	
// interval sending
// define what is selected
CASE eUploadType OF
	0: 	m_EnableChange_upload	:= FALSE;
		m_EnableInterval		:= TRUE;
		time_Interval			:= T#5M;
	1: 	m_EnableChange_upload	:= FALSE;
		m_EnableInterval		:= TRUE;
		time_Interval			:= T#1M;	
	2: 	m_EnableChange_upload	:= TRUE;
		m_EnableInterval		:= FALSE;
		time_Interval			:= T#5M;
	3: 	m_EnableChange_upload	:= TRUE;
		m_EnableInterval		:= TRUE;
		time_Interval			:= T#5M;	
	4: 	m_EnableChange_upload	:= TRUE;
		m_EnableInterval		:= TRUE;
		time_Interval			:= T#1M;	
END_CASE

// m_TriggerIntervalSend and m_EnableChange_upload used in line 997/996, 1011/1010 & 1606/1605

timer_Interval(IN:=NOT m_TriggerIntervalSend AND m_EnableInterval, PT:=time_Interval);
		
IF udiActiveNumberOfSymbol_ReadAds=udiNumberLoopFull_ReadAds AND iState_ReadAds>12 AND m_TriggerIntervalSend=TRUE  AND bFirstReadCycleDone_ReadAds THEN
	m_TriggerIntervalSend:=FALSE;
END_IF
IF (timer_interval.Q AND udiActiveNumberOfSymbol_ReadAds =0) THEN
	m_TriggerIntervalSend:=TRUE;
END_IF

END_FUNCTION_BLOCK

